// TIA Portal V20 export
FUNCTION_BLOCK "CallEquipment"   // FB64, LAD
TITLE = CallEquipment
// This block includes all general functions, checks and logik that is needed in the entire unit. E.g. general releases and system wide functionalities like air, pressure and power handling as well as general reaction to events.
// stored: IsIECCheckEnabled true, MemoryReserve 100, Namespace Unit1.Em6, SetENOAutomatically true
   VAR_INPUT
      ZoneOperationEnable { ExternalWritable := 'False'} : "LWONIK_typeSafetyZoneManualOperation";
   END_VAR
   VAR_IN_OUT
      unitStatus : "LAF_typeUnitStatus";   // Current unit status o be used in this EM
      emFeedback : "LUC_typeEmFeedback";   // Feedback of the EM to the Unit
      unitAlarmDB : "LAF_typeAlarms";   // Summarized EM Alarms for the Unit
   END_VAR
   VAR
      InstHotPressLeftSequence { ExternalWritable := 'False'} : "Unit1.Em6.Sequence_1_HotPressLeft";
      instHotPressLeftHomeJob1 { ExternalWritable := 'False'} : "LAF_SelectJob";
      instHotPressLeftLoadJob2 { ExternalWritable := 'False'} : "LAF_SelectJob";
      instHotPressLeftInspectionJob3 { ExternalWritable := 'False'} : "LAF_SelectJob";
      instHotPressLeftUnloadJob4 { ExternalWritable := 'False'} : "LAF_SelectJob";
      instCmHotPressLeftSafetyPin { ExternalWritable := 'False'} : "LBC_DigitalSignalCn";
      instCmHotPressLeftJRDetect { ExternalWritable := 'False'} : "LBC_DigitalSignalCn";
      instCmHotPressLeftStageLiftFrontUpDown { ExternalWritable := 'False'} : "LBC_TwoWayActuatorCn";
      instCmHotPressLeftStageLiftRearUpDown { ExternalWritable := 'False'} : "LBC_TwoWayActuatorCn";
      instCmHotPressLeftStageLiftAllUpDown { ExternalWritable := 'False'} : "LBC_TwoWayActuatorCn";
      instCmHotPressLeftTemperature { ExternalWritable := 'False'} : "LER_Heater";
      instCmHotPressLeftServoPress { ExternalWritable := 'False'} : "LER_ServoPress";
      instCmHotPressLeftHistroy { ExternalWritable := 'False'} : "LER_ServoPressHistory";
      instManageAlarms { ExternalWritable := 'False'} : "LAF_ManageAlarms";
      instEventsPFE { ExternalWritable := 'False'} : "Unit1.Em6.EventsPFE";
      statUnitStatus { ExternalWritable := 'False'} : "LAF_typeUnitStatus";   // Unit Status that is used in this project
   END_VAR
   VAR RETAIN
      statPartData { ExternalWritable := 'False'} : "LER_typePartData";
   END_VAR
   VAR
      statDataDelete { ExternalWritable := 'False'} : "LER_typePartData";
      statHistoryDeleteData { ExternalWritable := 'False'} : "LER_typeServoPressHistory";
      statClock { ExternalWritable := 'False'} : "LAF_typeGlobalClockMem";
      statTonTime { ExternalWritable := 'False'} : Array[0..999] of TON_TIME;
      statTofTime { ExternalWritable := 'False'} : Array[0..9] of TOF_TIME;
      statPulse { ExternalWritable := 'False'} : Array[0..999] of Bool;
      statNomalMode { ExternalWritable := 'False'} : Bool;
      statEnableManualCmds { ExternalWritable := 'False'} : Bool;
      statDoorOpenTemperature { ExternalWritable := 'False'} : "Safety.typeHotPressTempOk";
      statRunTemperature { ExternalWritable := 'False'} : Bool;
      "*** Interlock TwoWay ***" { S7_SetPoint := 'True'} : "LER_Axis_Homing";
      instCmHotPressLeftStageLiftFrontUpDownInterlock { S7_SetPoint := 'True'} : Array[0..2] of "LER_Actuator";
      instCmHotPressLeftStageLiftRearUpDownInterlock { S7_SetPoint := 'True'} : Array[0..2] of "LER_Actuator";
      instCmHotPressLeftStageLiftAllUpDownInterlock { S7_SetPoint := 'True'} : Array[0..2] of "LER_Actuator";
      HotPressLeftStageLiftFrontUpDown_Inpos : Array[0..2] of Struct
         "Int" : Array[1..10] of Bool;
      END_STRUCT;
      HotPressLeftStageLiftRearUpDown_Inpos : Array[0..2] of Struct
         "Int" : Array[1..10] of Bool;
      END_STRUCT;
      HotPressLeftStageLiftAllUpDown_Inpos : Array[0..2] of Struct
         "Int" : Array[1..10] of Bool;
      END_STRUCT;
      citi_Ptrig : Array[0..20] of Bool;
      citiTon : Array[0..20] of TON_TIME;
      citi : Time;
      citiTest : Array[0..20] of Bool;
      statReal : Array[0..9] of Real;
      instPFERecipe { S7_SetPoint := 'True'} : "Unit1.Em6.EventsPFE_Recipe";
   END_VAR
   VAR_TEMP
      tempRET_VAL : Array[0..99] of Int;
      tempScInProduction : Bool;   // Mode Production and StateComplete
      tempScNoProduction : Bool;   // Mode Manual and StateComplete
      tempPlaceReq : Bool;   // Request placing to TRPnPRight
      tempInspecReq : Bool;
      tempPickReq : Bool;   // Request Pick to TRPnPRight
   END_VAR
   VAR CONSTANT
      delayTime : Time := T#3s;
      TRUE : Bool := TRUE;
      FALSE : Bool := FALSE;
      NO_JOB : DInt;
      Stacker1 : Char := 'A';
      Stacker2 : Char := 'B';
   END_VAR
   VAR_TEMP   // added for the SCL form of the ladder/FBD networks
      _w1 : Bool;
      _w2 : Bool;
      _w3 : Bool;
      _w4 : Bool;
      _w5 : Bool;
      _w6 : Bool;
      _w7 : Bool;
   END_VAR
BEGIN

REGION Network 1: BLOCK INFO HEADER
   // (company) / (C) Copyright (year)
   // ---------------------------------------------------------------------------------
   // Title:                             (Title of this block)
   // Comment/Function: (that is implemented in the block)
   // Library/Family:           (that the source is dedicated to)
   // Author:                        (department / person in charge / contact)
   // Target System:          (test system with FW version)
   // Engineering:              TIA Portal (SW version)
   // Restrictions:               (OB types, etc.)
   // Requirements:           (hardware, technological package, etc.)
   // ---------------------------------------------------------------------------------
   // Change log table:
   // Version          | Date             | Signature      | Expert in charge  | Changes applied ------------------------|----------------------|-------------------------|--------------------------------|-----------------------
   // 001.000.000 | yyyy-mm-dd | 0x00000000 | (name of expert) | First released version
END_REGION

REGION Network 2: DESCRIPTION
   // This is a template block provided by the Automation Framework. It can be used to create an own project.
   // The Block Info Header is prepared to put in your own data.
   // Description of the block could be added here and the docu created by Code2Docu.
END_REGION

REGION Network 3: Simulation
   // If simulation is active on a global level, inherit this status and set simulation active in this unit also. Information is written to DB ControlNodes, from where it is distributed to the equipmemt modules.
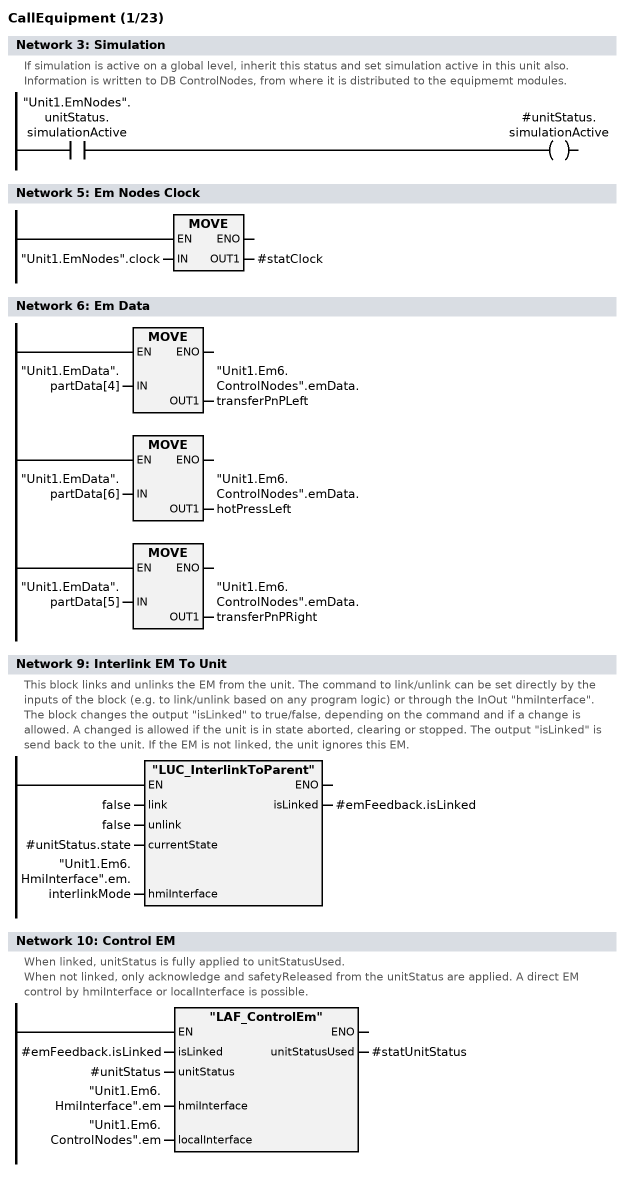
   RUNG wire#powerrail
      Contact( "Unit1.EmNodes".unitStatus.simulationActive )
      Coil( #unitStatus.simulationActive )
   END_RUNG
   // the same network as SCL:
   #unitStatus.simulationActive := "Unit1.EmNodes".unitStatus.simulationActive;
END_REGION

REGION Network 4: ******************** Unit Input ********************
END_REGION

REGION Network 5: Em Nodes Clock
   RUNG wire#powerrail
      Move(in := "Unit1.EmNodes".clock, out1 => #statClock)
   END_RUNG
   // the same network as SCL:
   #statClock := "Unit1.EmNodes".clock;
END_REGION

REGION Network 6: Em Data
   RUNG wire#powerrail
      Move(in := "Unit1.EmData".partData[4], out1 => "Unit1.Em6.ControlNodes".emData.transferPnPLeft)
   END_RUNG
   RUNG wire#powerrail
      Move(in := "Unit1.EmData".partData[6], out1 => "Unit1.Em6.ControlNodes".emData.hotPressLeft)
   END_RUNG
   RUNG wire#powerrail
      Move(in := "Unit1.EmData".partData[5], out1 => "Unit1.Em6.ControlNodes".emData.transferPnPRight)
   END_RUNG
   // the same network as SCL:
   "Unit1.Em6.ControlNodes".emData.transferPnPLeft := "Unit1.EmData".partData[4];
   "Unit1.Em6.ControlNodes".emData.hotPressLeft := "Unit1.EmData".partData[6];
   "Unit1.Em6.ControlNodes".emData.transferPnPRight := "Unit1.EmData".partData[5];
END_REGION

REGION Network 8: ******************** Equipment Control ********************
END_REGION

REGION Network 9: Interlink EM To Unit
   // This block links and unlinks the EM from the unit. The command to link/unlink can be set directly by the inputs of the block (e.g. to link/unlink based on any program logic) or through the InOut "hmiInterface". The block changes the output "isLinked" to true/false, depending on the command and if a change is allowed. A changed is allowed if the unit is in state aborted, clearing or stopped. The output "isLinked" is send back to the unit. If the EM is not linked, the unit ignores this EM.
   RUNG wire#powerrail
      "LUC_InterlinkToParent"(link := false, unlink := false, currentState := #unitStatus.state, hmiInterface := "Unit1.Em6.HmiInterface".em.interlinkMode, isLinked => #emFeedback.isLinked)
   END_RUNG
   // the same network as SCL:
   "LUC_InterlinkToParent"(link := false,
                           unlink := false,
                           currentState := #unitStatus.state,
                           hmiInterface := "Unit1.Em6.HmiInterface".em.interlinkMode,
                           isLinked => #emFeedback.isLinked);
END_REGION

REGION Network 10: Control EM
   // When linked, unitStatus is fully applied to unitStatusUsed.
   // When not linked, only acknowledge and safetyReleased from the unitStatus are applied. A direct EM control by hmiInterface or localInterface is possible.
   RUNG wire#powerrail
      "LAF_ControlEm"(isLinked := #emFeedback.isLinked, unitStatus := #unitStatus, hmiInterface := "Unit1.Em6.HmiInterface".em, localInterface := "Unit1.Em6.ControlNodes".em, unitStatusUsed => #statUnitStatus)
   END_RUNG
   // the same network as SCL:
   "LAF_ControlEm"(isLinked := #emFeedback.isLinked,
                   unitStatus := #unitStatus,
                   hmiInterface := "Unit1.Em6.HmiInterface".em,
                   localInterface := "Unit1.Em6.ControlNodes".em,
                   unitStatusUsed => #statUnitStatus);
END_REGION

REGION Network 11: EnableManualCmds
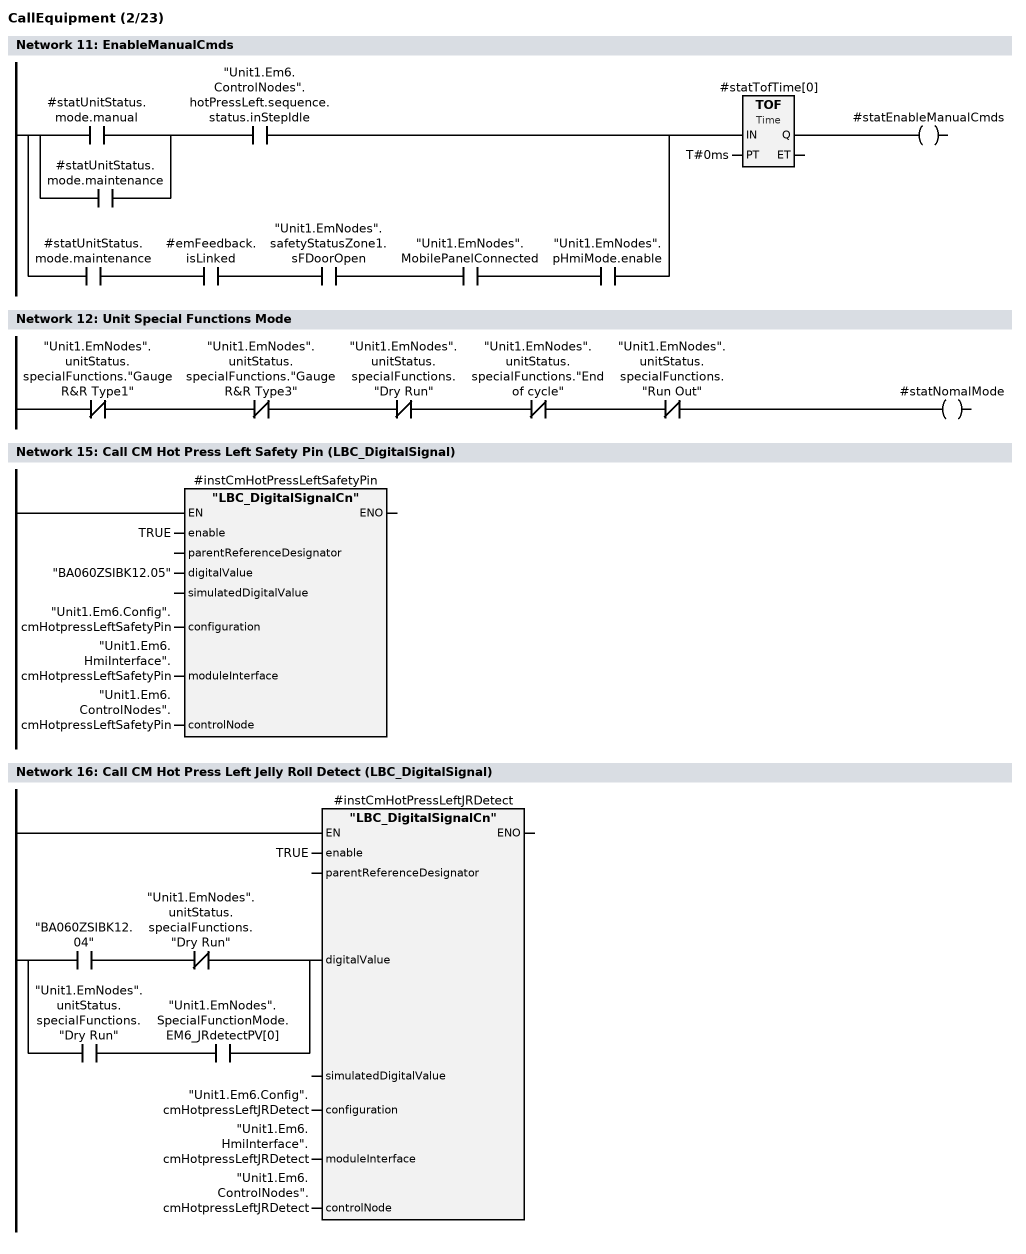
   RUNG wire#powerrail
      Contact( #statUnitStatus.mode.manual )
      wire#w1
      Contact( "Unit1.Em6.ControlNodes".hotPressLeft.sequence.status.inStepIdle )
      wire#w2
      { S7_Templates := "time_type := Time" } #statTofTime[0].TOF(pt := T#0ms, et =>)
      Coil( #statEnableManualCmds )
   END_RUNG
   RUNG wire#powerrail
      Contact( #statUnitStatus.mode.maintenance )
   END_RUNG wire#w1
   RUNG wire#powerrail
      Contact( #statUnitStatus.mode.maintenance )
      Contact( #emFeedback.isLinked )
      Contact( "Unit1.EmNodes".safetyStatusZone1.sFDoorOpen )
      Contact( "Unit1.EmNodes".MobilePanelConnected )
      Contact( "Unit1.EmNodes".pHmiMode.enable )
   END_RUNG wire#w2
   // the same network as SCL:
   #statTofTime[0].TOF(IN := ((#statUnitStatus.mode.manual OR #statUnitStatus.mode.maintenance) AND "Unit1.Em6.ControlNodes".hotPressLeft.sequence.status.inStepIdle) OR (#statUnitStatus.mode.maintenance AND #emFeedback.isLinked AND "Unit1.EmNodes".safetyStatusZone1.sFDoorOpen AND "Unit1.EmNodes".MobilePanelConnected AND "Unit1.EmNodes".pHmiMode.enable),
                       PT := T#0ms);
   #statEnableManualCmds := #statTofTime[0].Q;
END_REGION

REGION Network 12: Unit Special Functions Mode
   RUNG wire#powerrail
      I_Contact( "Unit1.EmNodes".unitStatus.specialFunctions."Gauge R&R Type1" )
      I_Contact( "Unit1.EmNodes".unitStatus.specialFunctions."Gauge R&R Type3" )
      I_Contact( "Unit1.EmNodes".unitStatus.specialFunctions."Dry Run" )
      I_Contact( "Unit1.EmNodes".unitStatus.specialFunctions."End of cycle" )
      I_Contact( "Unit1.EmNodes".unitStatus.specialFunctions."Run Out" )
      Coil( #statNomalMode )
   END_RUNG
   // the same network as SCL:
   #statNomalMode := NOT "Unit1.EmNodes".unitStatus.specialFunctions."Gauge R&R Type1" AND NOT "Unit1.EmNodes".unitStatus.specialFunctions."Gauge R&R Type3" AND NOT "Unit1.EmNodes".unitStatus.specialFunctions."Dry Run" AND NOT "Unit1.EmNodes".unitStatus.specialFunctions."End of cycle" AND NOT "Unit1.EmNodes".unitStatus.specialFunctions."Run Out";
END_REGION

REGION Network 14: ******************** Control Modules (Sensors) ********************
   // Call control modules that are sensors before the em logic (jobs and sequence), so that the latest value is used in the logic.
END_REGION

REGION Network 15: Call CM Hot Press Left Safety Pin (LBC_DigitalSignal)
   RUNG wire#powerrail
      #instCmHotPressLeftSafetyPin(enable := TRUE, parentReferenceDesignator :=, digitalValue := "BA060ZSIBK12.05", simulatedDigitalValue :=, configuration := "Unit1.Em6.Config".cmHotpressLeftSafetyPin, moduleInterface := "Unit1.Em6.HmiInterface".cmHotpressLeftSafetyPin, controlNode := "Unit1.Em6.ControlNodes".cmHotpressLeftSafetyPin)
   END_RUNG
   // the same network as SCL:
   #instCmHotPressLeftSafetyPin(enable := TRUE,   // "LBC_DigitalSignalCn"
                           digitalValue := "BA060ZSIBK12.05",
                           configuration := "Unit1.Em6.Config".cmHotpressLeftSafetyPin,
                           moduleInterface := "Unit1.Em6.HmiInterface".cmHotpressLeftSafetyPin,
                           controlNode := "Unit1.Em6.ControlNodes".cmHotpressLeftSafetyPin);
END_REGION

REGION Network 16: Call CM Hot Press Left Jelly Roll Detect (LBC_DigitalSignal)
   RUNG wire#powerrail
      #instCmHotPressLeftJRDetect(digitalValue := wire#w1, enable := TRUE, parentReferenceDesignator :=, simulatedDigitalValue :=, configuration := "Unit1.Em6.Config".cmHotpressLeftJRDetect, moduleInterface := "Unit1.Em6.HmiInterface".cmHotpressLeftJRDetect, controlNode := "Unit1.Em6.ControlNodes".cmHotpressLeftJRDetect)
   END_RUNG
   RUNG wire#powerrail
      Contact( "BA060ZSIBK12.04" )
      I_Contact( "Unit1.EmNodes".unitStatus.specialFunctions."Dry Run" )
   END_RUNG wire#w1
   RUNG wire#powerrail
      Contact( "Unit1.EmNodes".unitStatus.specialFunctions."Dry Run" )
      Contact( "Unit1.EmNodes".SpecialFunctionMode.EM6_JRdetectPV[0] )
   END_RUNG wire#w1
   // the same network as SCL:
   #instCmHotPressLeftJRDetect(enable := TRUE,   // "LBC_DigitalSignalCn"
                           digitalValue := ("BA060ZSIBK12.04" AND NOT "Unit1.EmNodes".unitStatus.specialFunctions."Dry Run") OR ("Unit1.EmNodes".unitStatus.specialFunctions."Dry Run" AND "Unit1.EmNodes".SpecialFunctionMode.EM6_JRdetectPV[0]),
                           configuration := "Unit1.Em6.Config".cmHotpressLeftJRDetect,
                           moduleInterface := "Unit1.Em6.HmiInterface".cmHotpressLeftJRDetect,
                           controlNode := "Unit1.Em6.ControlNodes".cmHotpressLeftJRDetect);
END_REGION

REGION Network 18: ******************** Equipment Logic ********************
END_REGION

REGION Network 19: Map Unit Status To Sequence Status
   // This block maps the unit status to the seuqnce status. Thus, it controls the sequence depending on the unit status. E.g. it sets the sequence to automatic when the unit state is in productions. This blocks work perfectly with the sequences provided in the AF. 
   // This typed block (MapUnitStatusToSequence) could be adjusted to specific application requirements or if other, user-defined sequences are used.
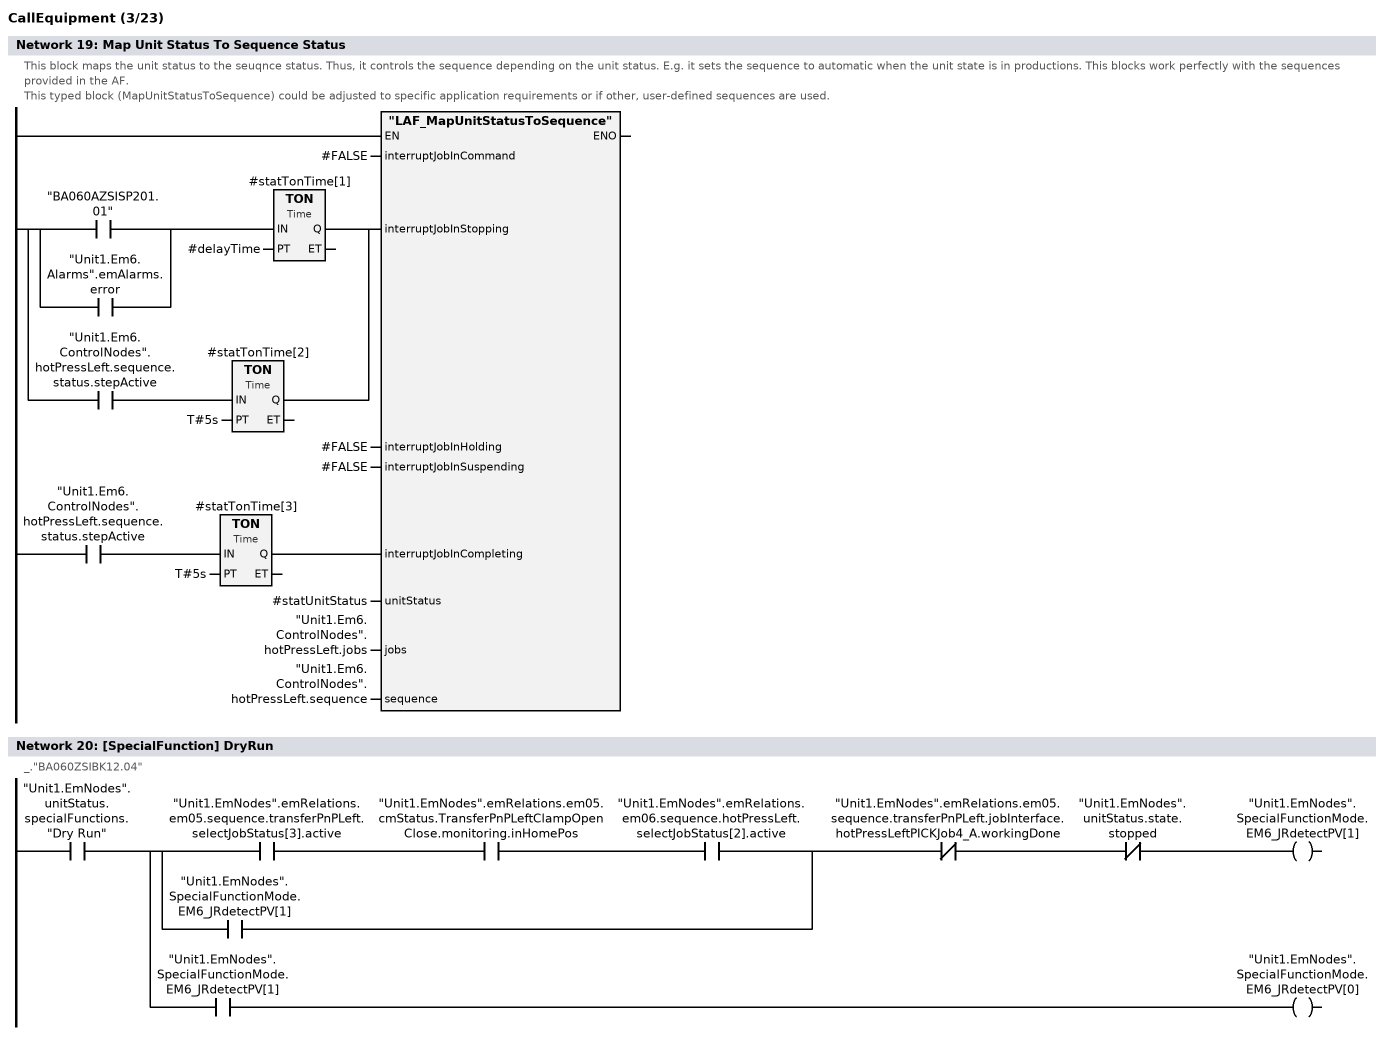
   RUNG wire#powerrail
      "LAF_MapUnitStatusToSequence"(interruptJobInStopping := wire#w2, interruptJobInCompleting := wire#w3, interruptJobInCommand := #FALSE, interruptJobInHolding := #FALSE, interruptJobInSuspending := #FALSE, unitStatus := #statUnitStatus, jobs := "Unit1.Em6.ControlNodes".hotPressLeft.jobs, sequence := "Unit1.Em6.ControlNodes".hotPressLeft.sequence)
   END_RUNG
   RUNG wire#powerrail
      Contact( "BA060AZSISP201.01" )
      wire#w1
      { S7_Templates := "time_type := Time" } #statTonTime[1].TON(pt := #delayTime, et =>)
   END_RUNG wire#w2
   RUNG wire#powerrail
      Contact( "Unit1.Em6.Alarms".emAlarms.error )
   END_RUNG wire#w1
   RUNG wire#powerrail
      Contact( "Unit1.Em6.ControlNodes".hotPressLeft.sequence.status.stepActive )
      { S7_Templates := "time_type := Time" } #statTonTime[2].TON(pt := T#5s, et =>)
   END_RUNG wire#w2
   RUNG wire#powerrail
      Contact( "Unit1.Em6.ControlNodes".hotPressLeft.sequence.status.stepActive )
      { S7_Templates := "time_type := Time" } #statTonTime[3].TON(pt := T#5s, et =>)
   END_RUNG wire#w3
   // the same network as SCL:
   #statTonTime[1].TON(IN := "BA060AZSISP201.01" OR "Unit1.Em6.Alarms".emAlarms.error, PT := #delayTime);
   #_w1 := #statTonTime[1].Q;
   #statTonTime[2].TON(IN := "Unit1.Em6.ControlNodes".hotPressLeft.sequence.status.stepActive, PT := T#5s);
   #_w2 := #_w1 OR #statTonTime[2].Q;
   #statTonTime[3].TON(IN := "Unit1.Em6.ControlNodes".hotPressLeft.sequence.status.stepActive, PT := T#5s);
   "LAF_MapUnitStatusToSequence"(interruptJobInCommand := #FALSE,
                           interruptJobInStopping := #_w2,
                           interruptJobInHolding := #FALSE,
                           interruptJobInSuspending := #FALSE,
                           interruptJobInCompleting := #statTonTime[3].Q,
                           unitStatus := #statUnitStatus,
                           jobs := "Unit1.Em6.ControlNodes".hotPressLeft.jobs,
                           sequence := "Unit1.Em6.ControlNodes".hotPressLeft.sequence);
END_REGION

REGION Network 20: [SpecialFunction] DryRun
   // _."BA060ZSIBK12.04"
   RUNG wire#powerrail
      Contact( "Unit1.EmNodes".unitStatus.specialFunctions."Dry Run" )
      wire#w1
      Contact( "Unit1.EmNodes".emRelations.em05.sequence.transferPnPLeft.selectJobStatus[3].active )
      Contact( "Unit1.EmNodes".emRelations.em05.cmStatus.TransferPnPLeftClampOpenClose.monitoring.inHomePos )
      Contact( "Unit1.EmNodes".emRelations.em06.sequence.hotPressLeft.selectJobStatus[2].active )
      wire#w2
      I_Contact( "Unit1.EmNodes".emRelations.em05.sequence.transferPnPLeft.jobInterface.hotPressLeftPICKJob4_A.workingDone )
      I_Contact( "Unit1.EmNodes".unitStatus.state.stopped )
      Coil( "Unit1.EmNodes".SpecialFunctionMode.EM6_JRdetectPV[1] )
   END_RUNG
   RUNG wire#w1
      Contact( "Unit1.EmNodes".SpecialFunctionMode.EM6_JRdetectPV[1] )
   END_RUNG wire#w2
   RUNG wire#w1
      Contact( "Unit1.EmNodes".SpecialFunctionMode.EM6_JRdetectPV[1] )
      Coil( "Unit1.EmNodes".SpecialFunctionMode.EM6_JRdetectPV[0] )
   END_RUNG
   // the same network as SCL:
   "Unit1.EmNodes".SpecialFunctionMode.EM6_JRdetectPV[1] := "Unit1.EmNodes".unitStatus.specialFunctions."Dry Run" AND (("Unit1.EmNodes".emRelations.em05.sequence.transferPnPLeft.selectJobStatus[3].active AND "Unit1.EmNodes".emRelations.em05.cmStatus.TransferPnPLeftClampOpenClose.monitoring.inHomePos AND "Unit1.EmNodes".emRelations.em06.sequence.hotPressLeft.selectJobStatus[2].active) OR "Unit1.EmNodes".SpecialFunctionMode.EM6_JRdetectPV[1]) AND NOT "Unit1.EmNodes".emRelations.em05.sequence.transferPnPLeft.jobInterface.hotPressLeftPICKJob4_A.workingDone AND NOT "Unit1.EmNodes".unitStatus.state.stopped;
   "Unit1.EmNodes".SpecialFunctionMode.EM6_JRdetectPV[0] := "Unit1.EmNodes".unitStatus.specialFunctions."Dry Run" AND "Unit1.EmNodes".SpecialFunctionMode.EM6_JRdetectPV[1];
END_REGION

REGION Network 22: [Job] Hot Press Left Select Job
   // Configure here when the jobs of the sequence should be started. More jobs could be added.
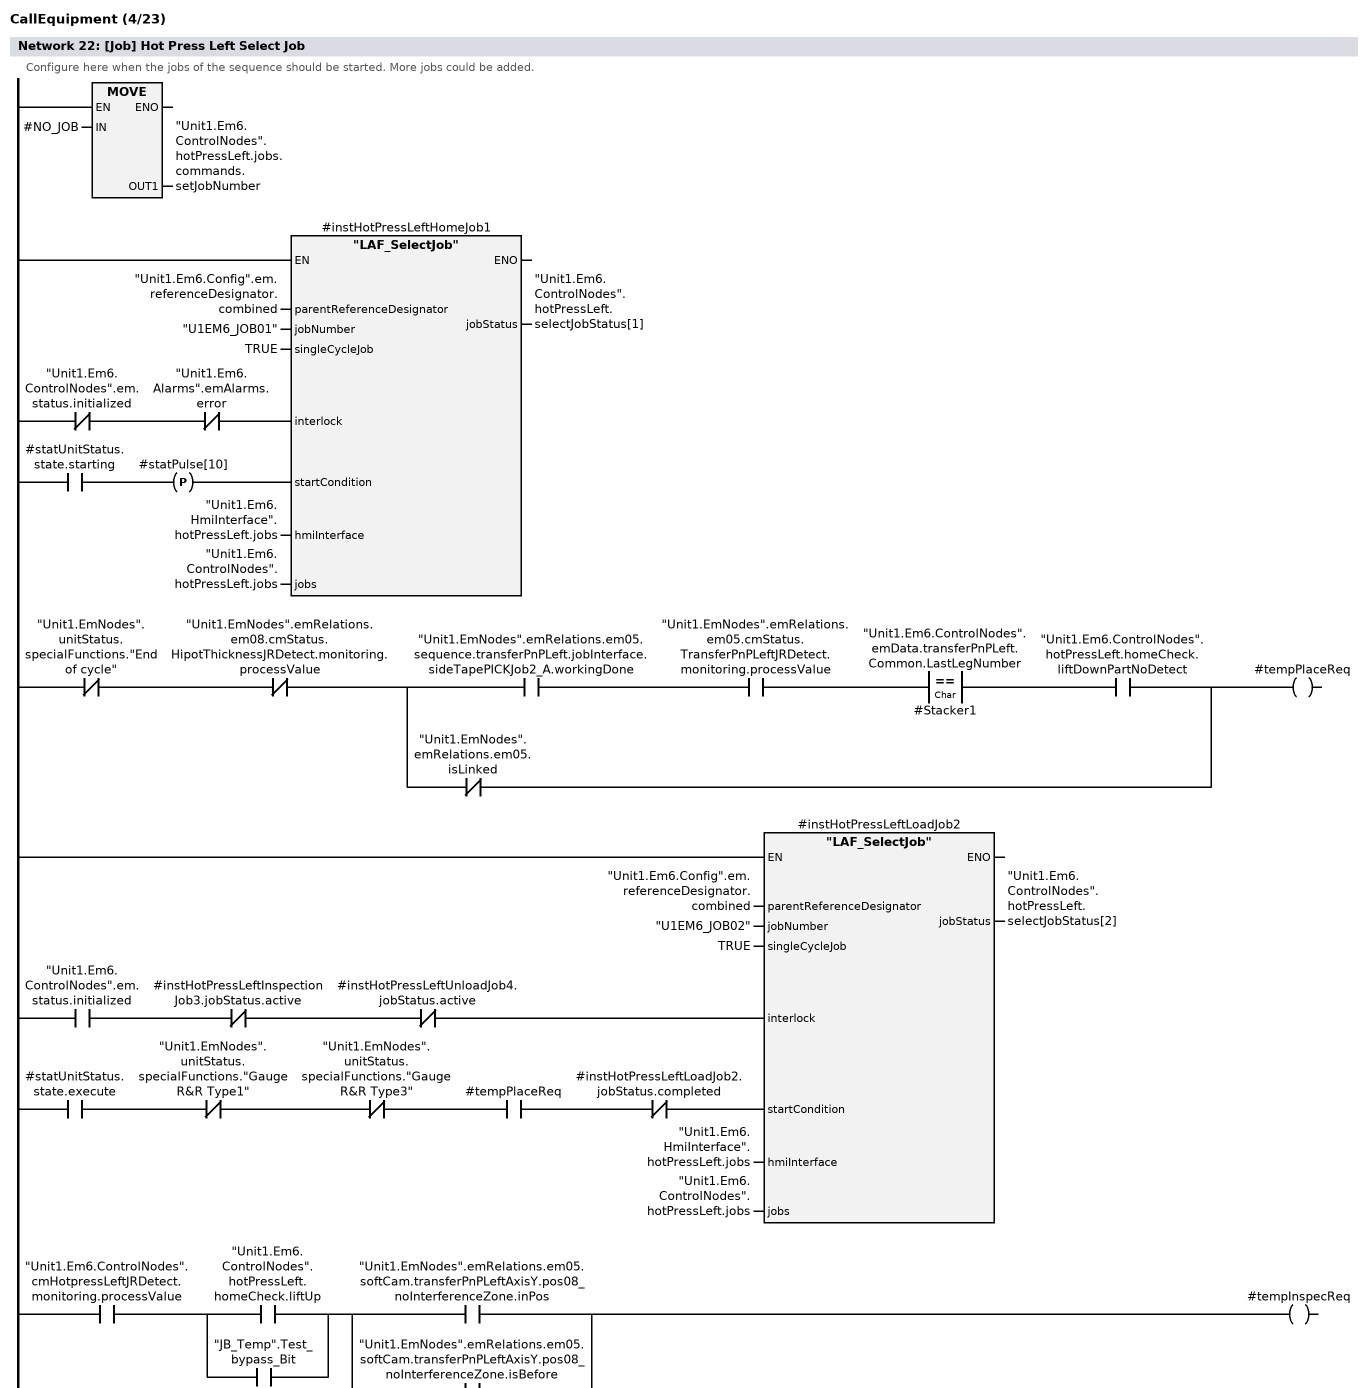
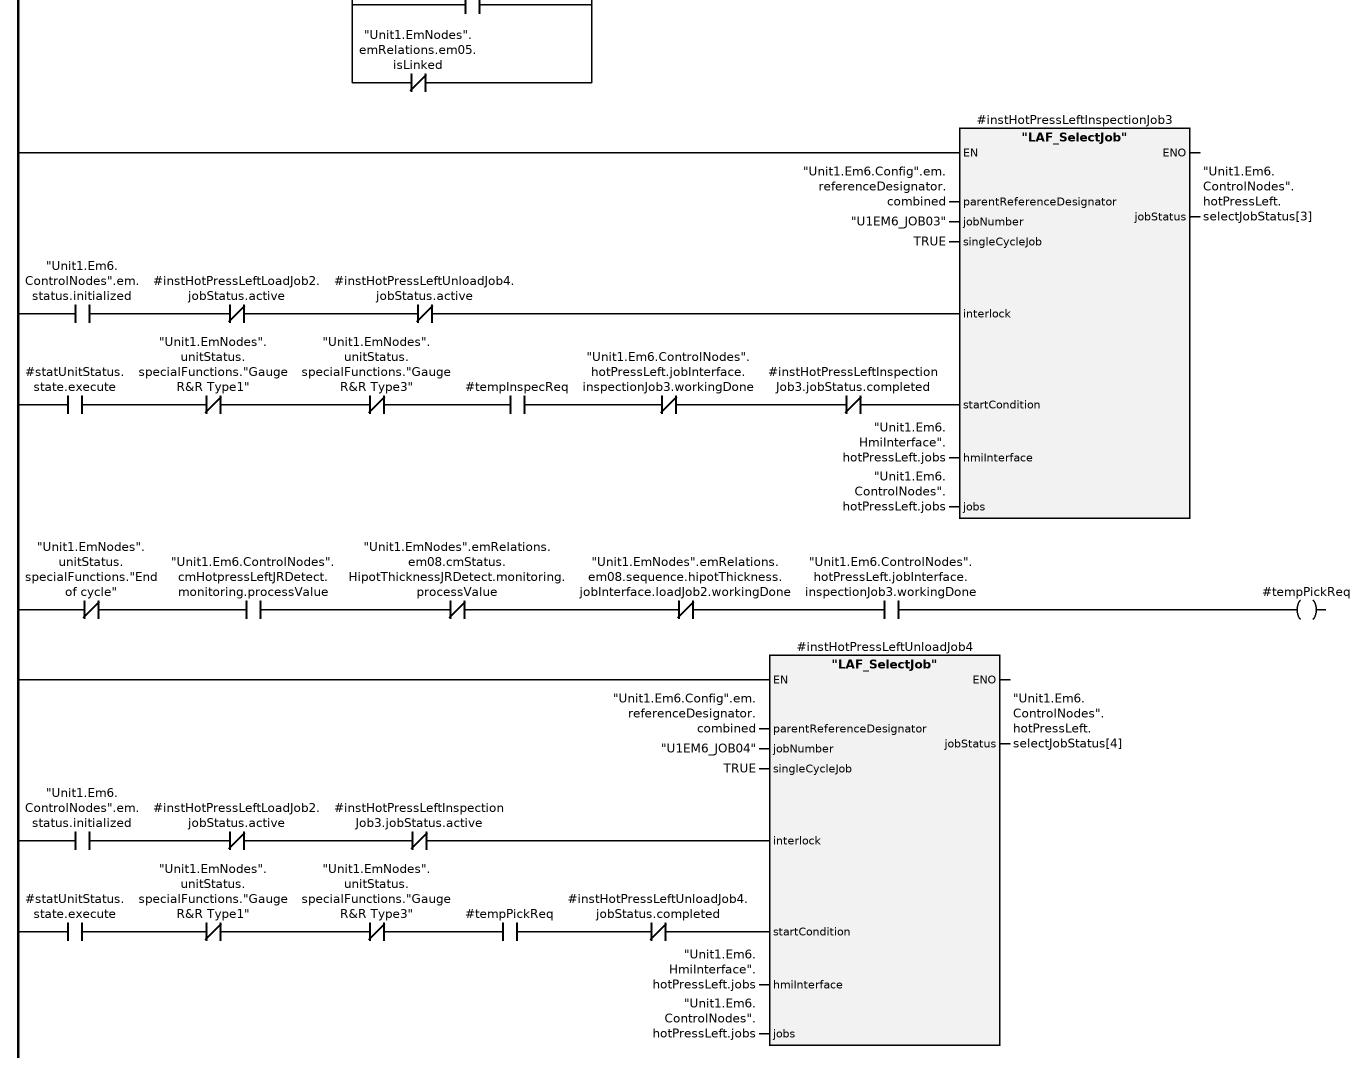
   RUNG wire#powerrail
      Move(in := #NO_JOB, out1 => "Unit1.Em6.ControlNodes".hotPressLeft.jobs.commands.setJobNumber)
   END_RUNG
   RUNG wire#powerrail
      #instHotPressLeftHomeJob1(interlock := wire#w1, startCondition := wire#w2, parentReferenceDesignator := "Unit1.Em6.Config".em.referenceDesignator.combined, jobNumber := "U1EM6_JOB01", singleCycleJob := TRUE, hmiInterface := "Unit1.Em6.HmiInterface".hotPressLeft.jobs, jobs := "Unit1.Em6.ControlNodes".hotPressLeft.jobs, jobStatus => "Unit1.Em6.ControlNodes".hotPressLeft.selectJobStatus[1])
   END_RUNG
   RUNG wire#powerrail
      I_Contact( "Unit1.Em6.ControlNodes".em.status.initialized )
      I_Contact( "Unit1.Em6.Alarms".emAlarms.error )
   END_RUNG wire#w1
   RUNG wire#powerrail
      Contact( #statUnitStatus.state.starting )
      P_Trig( #statPulse[10] )
   END_RUNG wire#w2
   RUNG wire#powerrail
      I_Contact( "Unit1.EmNodes".unitStatus.specialFunctions."End of cycle" )
      I_Contact( "Unit1.EmNodes".emRelations.em08.cmStatus.HipotThicknessJRDetect.monitoring.processValue )
      wire#w3
      Contact( "Unit1.EmNodes".emRelations.em05.sequence.transferPnPLeft.jobInterface.sideTapePICKJob2_A.workingDone )
      Contact( "Unit1.EmNodes".emRelations.em05.cmStatus.TransferPnPLeftJRDetect.monitoring.processValue )
      { S7_Templates := "SrcType := Char" } EQ_Contact(in1 := "Unit1.Em6.ControlNodes".emData.transferPnPLeft.Common.LastLegNumber, in2 := #Stacker1)
      Contact( "Unit1.Em6.ControlNodes".hotPressLeft.homeCheck.liftDownPartNoDetect )
      wire#w4
      Coil( #tempPlaceReq )
   END_RUNG
   RUNG wire#w3
      I_Contact( "Unit1.EmNodes".emRelations.em05.isLinked )
   END_RUNG wire#w4
   RUNG wire#powerrail
      #instHotPressLeftLoadJob2(interlock := wire#w5, startCondition := wire#w6, parentReferenceDesignator := "Unit1.Em6.Config".em.referenceDesignator.combined, jobNumber := "U1EM6_JOB02", singleCycleJob := TRUE, hmiInterface := "Unit1.Em6.HmiInterface".hotPressLeft.jobs, jobs := "Unit1.Em6.ControlNodes".hotPressLeft.jobs, jobStatus => "Unit1.Em6.ControlNodes".hotPressLeft.selectJobStatus[2])
   END_RUNG
   RUNG wire#powerrail
      Contact( "Unit1.Em6.ControlNodes".em.status.initialized )
      I_Contact( #instHotPressLeftInspectionJob3.jobStatus.active )
      I_Contact( #instHotPressLeftUnloadJob4.jobStatus.active )
   END_RUNG wire#w5
   RUNG wire#powerrail
      Contact( #statUnitStatus.state.execute )
      I_Contact( "Unit1.EmNodes".unitStatus.specialFunctions."Gauge R&R Type1" )
      I_Contact( "Unit1.EmNodes".unitStatus.specialFunctions."Gauge R&R Type3" )
      Contact( #tempPlaceReq )
      I_Contact( #instHotPressLeftLoadJob2.jobStatus.completed )
   END_RUNG wire#w6
   RUNG wire#powerrail
      Contact( "Unit1.Em6.ControlNodes".cmHotpressLeftJRDetect.monitoring.processValue )
      wire#w7
      Contact( "Unit1.Em6.ControlNodes".hotPressLeft.homeCheck.liftUp )
      wire#w8
      Contact( "Unit1.EmNodes".emRelations.em05.softCam.transferPnPLeftAxisY.pos08_noInterferenceZone.inPos )
      wire#w9
      Coil( #tempInspecReq )
   END_RUNG
   RUNG wire#w7
      Contact( "JB_Temp".Test_bypass_Bit )
   END_RUNG wire#w8
   RUNG wire#w8
      Contact( "Unit1.EmNodes".emRelations.em05.softCam.transferPnPLeftAxisY.pos08_noInterferenceZone.isBefore )
   END_RUNG wire#w9
   RUNG wire#w8
      I_Contact( "Unit1.EmNodes".emRelations.em05.isLinked )
   END_RUNG wire#w9
   RUNG wire#powerrail
      #instHotPressLeftInspectionJob3(interlock := wire#w10, startCondition := wire#w11, parentReferenceDesignator := "Unit1.Em6.Config".em.referenceDesignator.combined, jobNumber := "U1EM6_JOB03", singleCycleJob := TRUE, hmiInterface := "Unit1.Em6.HmiInterface".hotPressLeft.jobs, jobs := "Unit1.Em6.ControlNodes".hotPressLeft.jobs, jobStatus => "Unit1.Em6.ControlNodes".hotPressLeft.selectJobStatus[3])
   END_RUNG
   RUNG wire#powerrail
      Contact( "Unit1.Em6.ControlNodes".em.status.initialized )
      I_Contact( #instHotPressLeftLoadJob2.jobStatus.active )
      I_Contact( #instHotPressLeftUnloadJob4.jobStatus.active )
   END_RUNG wire#w10
   RUNG wire#powerrail
      Contact( #statUnitStatus.state.execute )
      I_Contact( "Unit1.EmNodes".unitStatus.specialFunctions."Gauge R&R Type1" )
      I_Contact( "Unit1.EmNodes".unitStatus.specialFunctions."Gauge R&R Type3" )
      Contact( #tempInspecReq )
      I_Contact( "Unit1.Em6.ControlNodes".hotPressLeft.jobInterface.inspectionJob3.workingDone )
      I_Contact( #instHotPressLeftInspectionJob3.jobStatus.completed )
   END_RUNG wire#w11
   RUNG wire#powerrail
      I_Contact( "Unit1.EmNodes".unitStatus.specialFunctions."End of cycle" )
      Contact( "Unit1.Em6.ControlNodes".cmHotpressLeftJRDetect.monitoring.processValue )
      I_Contact( "Unit1.EmNodes".emRelations.em08.cmStatus.HipotThicknessJRDetect.monitoring.processValue )
      I_Contact( "Unit1.EmNodes".emRelations.em08.sequence.hipotThickness.jobInterface.loadJob2.workingDone )
      Contact( "Unit1.Em6.ControlNodes".hotPressLeft.jobInterface.inspectionJob3.workingDone )
      Coil( #tempPickReq )
   END_RUNG
   RUNG wire#powerrail
      #instHotPressLeftUnloadJob4(interlock := wire#w12, startCondition := wire#w13, parentReferenceDesignator := "Unit1.Em6.Config".em.referenceDesignator.combined, jobNumber := "U1EM6_JOB04", singleCycleJob := TRUE, hmiInterface := "Unit1.Em6.HmiInterface".hotPressLeft.jobs, jobs := "Unit1.Em6.ControlNodes".hotPressLeft.jobs, jobStatus => "Unit1.Em6.ControlNodes".hotPressLeft.selectJobStatus[4])
   END_RUNG
   RUNG wire#powerrail
      Contact( "Unit1.Em6.ControlNodes".em.status.initialized )
      I_Contact( #instHotPressLeftLoadJob2.jobStatus.active )
      I_Contact( #instHotPressLeftInspectionJob3.jobStatus.active )
   END_RUNG wire#w12
   RUNG wire#powerrail
      Contact( #statUnitStatus.state.execute )
      I_Contact( "Unit1.EmNodes".unitStatus.specialFunctions."Gauge R&R Type1" )
      I_Contact( "Unit1.EmNodes".unitStatus.specialFunctions."Gauge R&R Type3" )
      Contact( #tempPickReq )
      I_Contact( #instHotPressLeftUnloadJob4.jobStatus.completed )
   END_RUNG wire#w13
   // the same network as SCL:
   "Unit1.Em6.ControlNodes".hotPressLeft.jobs.commands.setJobNumber := #NO_JOB;
   #_w1 := #statUnitStatus.state.starting AND NOT #statPulse[10];   // rising edge
   #statPulse[10] := #statUnitStatus.state.starting;
   #instHotPressLeftHomeJob1(parentReferenceDesignator := "Unit1.Em6.Config".em.referenceDesignator.combined,   // "LAF_SelectJob"
                           jobNumber := "U1EM6_JOB01",
                           singleCycleJob := TRUE,
                           interlock := NOT "Unit1.Em6.ControlNodes".em.status.initialized AND NOT "Unit1.Em6.Alarms".emAlarms.error,
                           startCondition := #_w1,
                           hmiInterface := "Unit1.Em6.HmiInterface".hotPressLeft.jobs,
                           jobs := "Unit1.Em6.ControlNodes".hotPressLeft.jobs,
                           jobStatus => "Unit1.Em6.ControlNodes".hotPressLeft.selectJobStatus[1]);
   #tempPlaceReq := NOT "Unit1.EmNodes".unitStatus.specialFunctions."End of cycle" AND NOT "Unit1.EmNodes".emRelations.em08.cmStatus.HipotThicknessJRDetect.monitoring.processValue AND (("Unit1.EmNodes".emRelations.em05.sequence.transferPnPLeft.jobInterface.sideTapePICKJob2_A.workingDone AND "Unit1.EmNodes".emRelations.em05.cmStatus.TransferPnPLeftJRDetect.monitoring.processValue AND ("Unit1.Em6.ControlNodes".emData.transferPnPLeft.Common.LastLegNumber = #Stacker1) AND "Unit1.Em6.ControlNodes".hotPressLeft.homeCheck.liftDownPartNoDetect) OR NOT "Unit1.EmNodes".emRelations.em05.isLinked);
   #instHotPressLeftLoadJob2(parentReferenceDesignator := "Unit1.Em6.Config".em.referenceDesignator.combined,   // "LAF_SelectJob"
                           jobNumber := "U1EM6_JOB02",
                           singleCycleJob := TRUE,
                           interlock := "Unit1.Em6.ControlNodes".em.status.initialized AND NOT #instHotPressLeftInspectionJob3.jobStatus.active AND NOT #instHotPressLeftUnloadJob4.jobStatus.active,
                           startCondition := #statUnitStatus.state.execute AND NOT "Unit1.EmNodes".unitStatus.specialFunctions."Gauge R&R Type1" AND NOT "Unit1.EmNodes".unitStatus.specialFunctions."Gauge R&R Type3" AND #tempPlaceReq AND NOT #instHotPressLeftLoadJob2.jobStatus.completed,
                           hmiInterface := "Unit1.Em6.HmiInterface".hotPressLeft.jobs,
                           jobs := "Unit1.Em6.ControlNodes".hotPressLeft.jobs,
                           jobStatus => "Unit1.Em6.ControlNodes".hotPressLeft.selectJobStatus[2]);
   #tempInspecReq := "Unit1.Em6.ControlNodes".cmHotpressLeftJRDetect.monitoring.processValue AND ("Unit1.Em6.ControlNodes".hotPressLeft.homeCheck.liftUp OR "JB_Temp".Test_bypass_Bit) AND ("Unit1.EmNodes".emRelations.em05.softCam.transferPnPLeftAxisY.pos08_noInterferenceZone.inPos OR "Unit1.EmNodes".emRelations.em05.softCam.transferPnPLeftAxisY.pos08_noInterferenceZone.isBefore OR NOT "Unit1.EmNodes".emRelations.em05.isLinked);
   #instHotPressLeftInspectionJob3(parentReferenceDesignator := "Unit1.Em6.Config".em.referenceDesignator.combined,   // "LAF_SelectJob"
                           jobNumber := "U1EM6_JOB03",
                           singleCycleJob := TRUE,
                           interlock := "Unit1.Em6.ControlNodes".em.status.initialized AND NOT #instHotPressLeftLoadJob2.jobStatus.active AND NOT #instHotPressLeftUnloadJob4.jobStatus.active,
                           startCondition := #statUnitStatus.state.execute AND NOT "Unit1.EmNodes".unitStatus.specialFunctions."Gauge R&R Type1" AND NOT "Unit1.EmNodes".unitStatus.specialFunctions."Gauge R&R Type3" AND #tempInspecReq AND NOT "Unit1.Em6.ControlNodes".hotPressLeft.jobInterface.inspectionJob3.workingDone AND NOT #instHotPressLeftInspectionJob3.jobStatus.completed,
                           hmiInterface := "Unit1.Em6.HmiInterface".hotPressLeft.jobs,
                           jobs := "Unit1.Em6.ControlNodes".hotPressLeft.jobs,
                           jobStatus => "Unit1.Em6.ControlNodes".hotPressLeft.selectJobStatus[3]);
   #tempPickReq := NOT "Unit1.EmNodes".unitStatus.specialFunctions."End of cycle" AND "Unit1.Em6.ControlNodes".cmHotpressLeftJRDetect.monitoring.processValue AND NOT "Unit1.EmNodes".emRelations.em08.cmStatus.HipotThicknessJRDetect.monitoring.processValue AND NOT "Unit1.EmNodes".emRelations.em08.sequence.hipotThickness.jobInterface.loadJob2.workingDone AND "Unit1.Em6.ControlNodes".hotPressLeft.jobInterface.inspectionJob3.workingDone;
   #instHotPressLeftUnloadJob4(parentReferenceDesignator := "Unit1.Em6.Config".em.referenceDesignator.combined,   // "LAF_SelectJob"
                           jobNumber := "U1EM6_JOB04",
                           singleCycleJob := TRUE,
                           interlock := "Unit1.Em6.ControlNodes".em.status.initialized AND NOT #instHotPressLeftLoadJob2.jobStatus.active AND NOT #instHotPressLeftInspectionJob3.jobStatus.active,
                           startCondition := #statUnitStatus.state.execute AND NOT "Unit1.EmNodes".unitStatus.specialFunctions."Gauge R&R Type1" AND NOT "Unit1.EmNodes".unitStatus.specialFunctions."Gauge R&R Type3" AND #tempPickReq AND NOT #instHotPressLeftUnloadJob4.jobStatus.completed,
                           hmiInterface := "Unit1.Em6.HmiInterface".hotPressLeft.jobs,
                           jobs := "Unit1.Em6.ControlNodes".hotPressLeft.jobs,
                           jobStatus => "Unit1.Em6.ControlNodes".hotPressLeft.selectJobStatus[4]);
END_REGION

REGION Network 23: Hot Press left Job Interface [Loading]
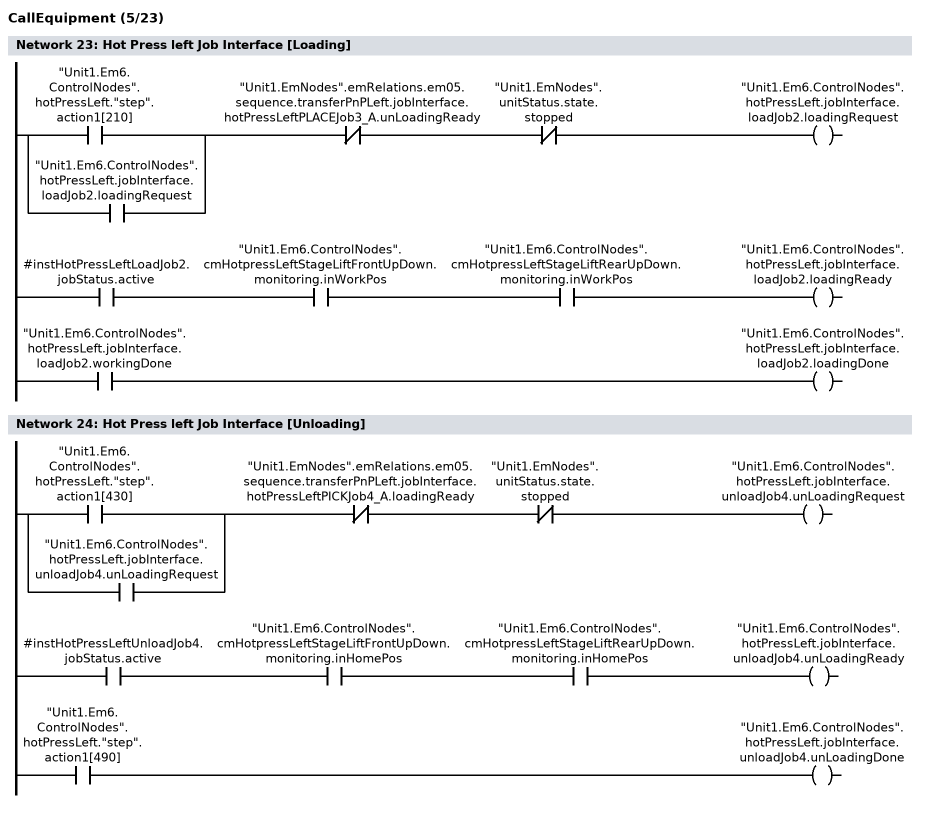
   RUNG wire#powerrail
      Contact( "Unit1.Em6.ControlNodes".hotPressLeft."step".action1[210] )
      wire#w1
      I_Contact( "Unit1.EmNodes".emRelations.em05.sequence.transferPnPLeft.jobInterface.hotPressLeftPLACEJob3_A.unLoadingReady )
      I_Contact( "Unit1.EmNodes".unitStatus.state.stopped )
      Coil( "Unit1.Em6.ControlNodes".hotPressLeft.jobInterface.loadJob2.loadingRequest )
   END_RUNG
   RUNG wire#powerrail
      Contact( "Unit1.Em6.ControlNodes".hotPressLeft.jobInterface.loadJob2.loadingRequest )
   END_RUNG wire#w1
   RUNG wire#powerrail
      Contact( #instHotPressLeftLoadJob2.jobStatus.active )
      Contact( "Unit1.Em6.ControlNodes".cmHotpressLeftStageLiftFrontUpDown.monitoring.inWorkPos )
      Contact( "Unit1.Em6.ControlNodes".cmHotpressLeftStageLiftRearUpDown.monitoring.inWorkPos )
      Coil( "Unit1.Em6.ControlNodes".hotPressLeft.jobInterface.loadJob2.loadingReady )
   END_RUNG
   RUNG wire#powerrail
      Contact( "Unit1.Em6.ControlNodes".hotPressLeft.jobInterface.loadJob2.workingDone )
      Coil( "Unit1.Em6.ControlNodes".hotPressLeft.jobInterface.loadJob2.loadingDone )
   END_RUNG
   // the same network as SCL:
   "Unit1.Em6.ControlNodes".hotPressLeft.jobInterface.loadJob2.loadingRequest := ("Unit1.Em6.ControlNodes".hotPressLeft."step".action1[210] OR "Unit1.Em6.ControlNodes".hotPressLeft.jobInterface.loadJob2.loadingRequest) AND NOT "Unit1.EmNodes".emRelations.em05.sequence.transferPnPLeft.jobInterface.hotPressLeftPLACEJob3_A.unLoadingReady AND NOT "Unit1.EmNodes".unitStatus.state.stopped;
   "Unit1.Em6.ControlNodes".hotPressLeft.jobInterface.loadJob2.loadingReady := #instHotPressLeftLoadJob2.jobStatus.active AND "Unit1.Em6.ControlNodes".cmHotpressLeftStageLiftFrontUpDown.monitoring.inWorkPos AND "Unit1.Em6.ControlNodes".cmHotpressLeftStageLiftRearUpDown.monitoring.inWorkPos;
   "Unit1.Em6.ControlNodes".hotPressLeft.jobInterface.loadJob2.loadingDone := "Unit1.Em6.ControlNodes".hotPressLeft.jobInterface.loadJob2.workingDone;
END_REGION

REGION Network 24: Hot Press left Job Interface [Unloading]
   RUNG wire#powerrail
      Contact( "Unit1.Em6.ControlNodes".hotPressLeft."step".action1[430] )
      wire#w1
      I_Contact( "Unit1.EmNodes".emRelations.em05.sequence.transferPnPLeft.jobInterface.hotPressLeftPICKJob4_A.loadingReady )
      I_Contact( "Unit1.EmNodes".unitStatus.state.stopped )
      Coil( "Unit1.Em6.ControlNodes".hotPressLeft.jobInterface.unloadJob4.unLoadingRequest )
   END_RUNG
   RUNG wire#powerrail
      Contact( "Unit1.Em6.ControlNodes".hotPressLeft.jobInterface.unloadJob4.unLoadingRequest )
   END_RUNG wire#w1
   RUNG wire#powerrail
      Contact( #instHotPressLeftUnloadJob4.jobStatus.active )
      Contact( "Unit1.Em6.ControlNodes".cmHotpressLeftStageLiftFrontUpDown.monitoring.inHomePos )
      Contact( "Unit1.Em6.ControlNodes".cmHotpressLeftStageLiftRearUpDown.monitoring.inHomePos )
      Coil( "Unit1.Em6.ControlNodes".hotPressLeft.jobInterface.unloadJob4.unLoadingReady )
   END_RUNG
   RUNG wire#powerrail
      Contact( "Unit1.Em6.ControlNodes".hotPressLeft."step".action1[490] )
      Coil( "Unit1.Em6.ControlNodes".hotPressLeft.jobInterface.unloadJob4.unLoadingDone )
   END_RUNG
   // the same network as SCL:
   "Unit1.Em6.ControlNodes".hotPressLeft.jobInterface.unloadJob4.unLoadingRequest := ("Unit1.Em6.ControlNodes".hotPressLeft."step".action1[430] OR "Unit1.Em6.ControlNodes".hotPressLeft.jobInterface.unloadJob4.unLoadingRequest) AND NOT "Unit1.EmNodes".emRelations.em05.sequence.transferPnPLeft.jobInterface.hotPressLeftPICKJob4_A.loadingReady AND NOT "Unit1.EmNodes".unitStatus.state.stopped;
   "Unit1.Em6.ControlNodes".hotPressLeft.jobInterface.unloadJob4.unLoadingReady := #instHotPressLeftUnloadJob4.jobStatus.active AND "Unit1.Em6.ControlNodes".cmHotpressLeftStageLiftFrontUpDown.monitoring.inHomePos AND "Unit1.Em6.ControlNodes".cmHotpressLeftStageLiftRearUpDown.monitoring.inHomePos;
   "Unit1.Em6.ControlNodes".hotPressLeft.jobInterface.unloadJob4.unLoadingDone := "Unit1.Em6.ControlNodes".hotPressLeft."step".action1[490];
END_REGION

REGION Network 25: Hot Press Left Job Interface Working Done
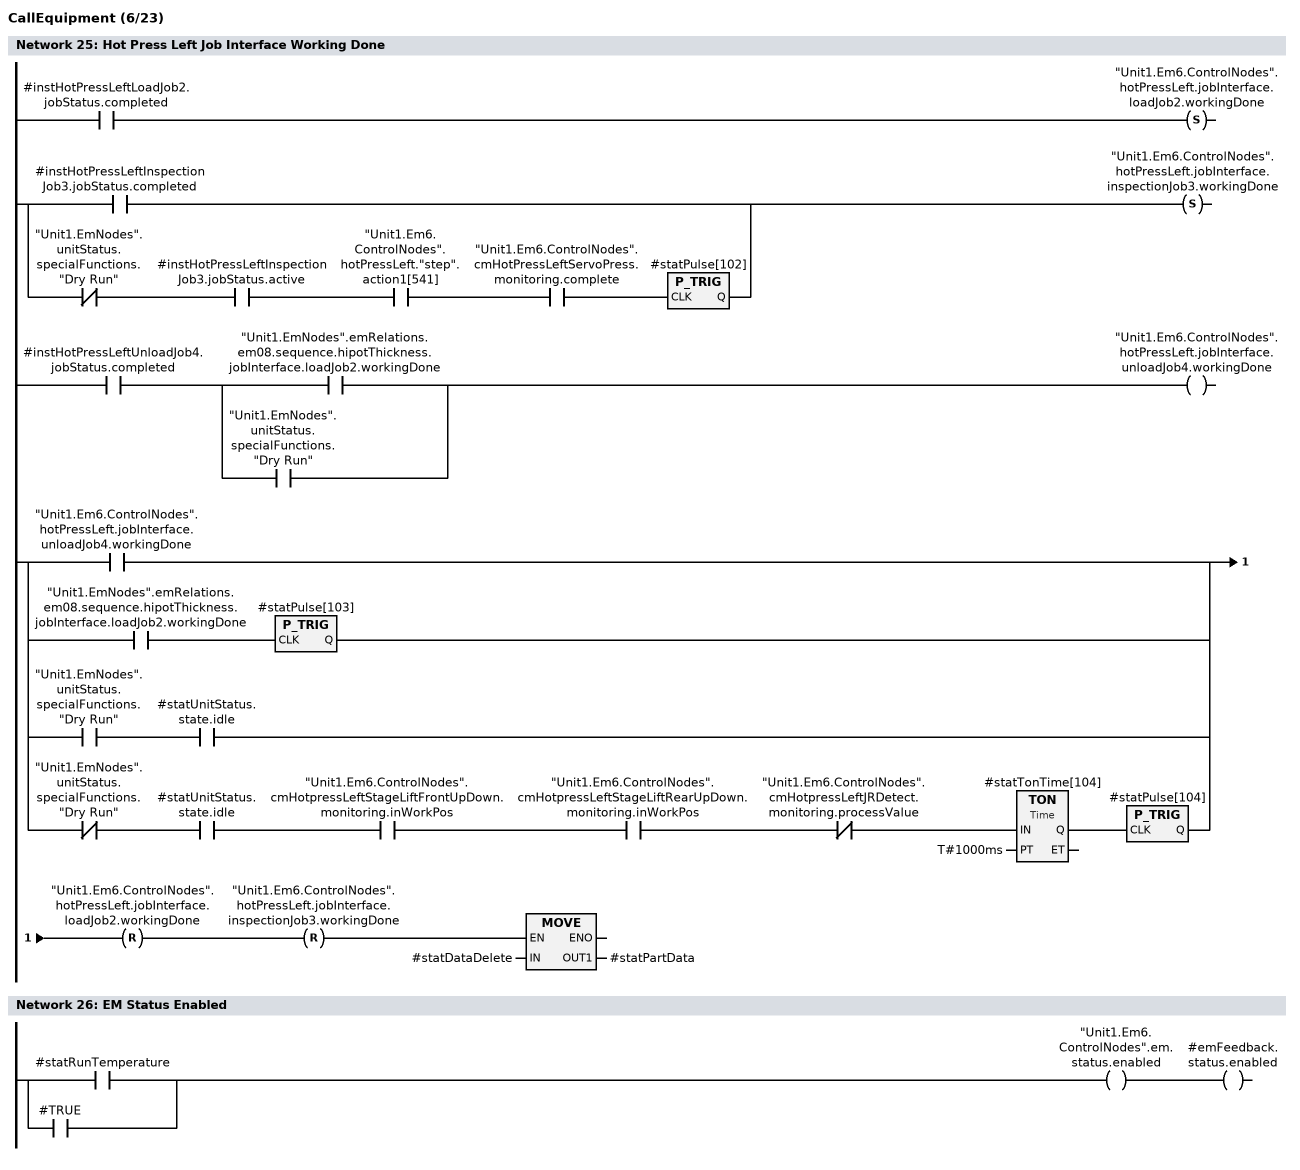
   RUNG wire#powerrail
      Contact( #instHotPressLeftLoadJob2.jobStatus.completed )
      S_Coil( "Unit1.Em6.ControlNodes".hotPressLeft.jobInterface.loadJob2.workingDone )
   END_RUNG
   RUNG wire#powerrail
      Contact( #instHotPressLeftInspectionJob3.jobStatus.completed )
      wire#w1
      S_Coil( "Unit1.Em6.ControlNodes".hotPressLeft.jobInterface.inspectionJob3.workingDone )
   END_RUNG
   RUNG wire#powerrail
      I_Contact( "Unit1.EmNodes".unitStatus.specialFunctions."Dry Run" )
      Contact( #instHotPressLeftInspectionJob3.jobStatus.active )
      Contact( "Unit1.Em6.ControlNodes".hotPressLeft."step".action1[541] )
      Contact( "Unit1.Em6.ControlNodes".cmHotPressLeftServoPress.monitoring.complete )
      P_Trig( #statPulse[102] )
   END_RUNG wire#w1
   RUNG wire#powerrail
      Contact( #instHotPressLeftUnloadJob4.jobStatus.completed )
      wire#w2
      Contact( "Unit1.EmNodes".emRelations.em08.sequence.hipotThickness.jobInterface.loadJob2.workingDone )
      wire#w3
      Coil( "Unit1.Em6.ControlNodes".hotPressLeft.jobInterface.unloadJob4.workingDone )
   END_RUNG
   RUNG wire#w2
      Contact( "Unit1.EmNodes".unitStatus.specialFunctions."Dry Run" )
   END_RUNG wire#w3
   RUNG wire#powerrail
      Contact( "Unit1.Em6.ControlNodes".hotPressLeft.jobInterface.unloadJob4.workingDone )
      wire#w4
      R_Coil( "Unit1.Em6.ControlNodes".hotPressLeft.jobInterface.loadJob2.workingDone )
      R_Coil( "Unit1.Em6.ControlNodes".hotPressLeft.jobInterface.inspectionJob3.workingDone )
      Move(in := #statDataDelete, out1 => #statPartData)
   END_RUNG
   RUNG wire#powerrail
      Contact( "Unit1.EmNodes".emRelations.em08.sequence.hipotThickness.jobInterface.loadJob2.workingDone )
      P_Trig( #statPulse[103] )
   END_RUNG wire#w4
   RUNG wire#powerrail
      Contact( "Unit1.EmNodes".unitStatus.specialFunctions."Dry Run" )
      Contact( #statUnitStatus.state.idle )
   END_RUNG wire#w4
   RUNG wire#powerrail
      I_Contact( "Unit1.EmNodes".unitStatus.specialFunctions."Dry Run" )
      Contact( #statUnitStatus.state.idle )
      Contact( "Unit1.Em6.ControlNodes".cmHotpressLeftStageLiftFrontUpDown.monitoring.inWorkPos )
      Contact( "Unit1.Em6.ControlNodes".cmHotpressLeftStageLiftRearUpDown.monitoring.inWorkPos )
      I_Contact( "Unit1.Em6.ControlNodes".cmHotpressLeftJRDetect.monitoring.processValue )
      { S7_Templates := "time_type := Time" } #statTonTime[104].TON(pt := T#1000ms, et =>)
      P_Trig( #statPulse[104] )
   END_RUNG wire#w4
   // the same network as SCL:
   IF #instHotPressLeftLoadJob2.jobStatus.completed THEN
       "Unit1.Em6.ControlNodes".hotPressLeft.jobInterface.loadJob2.workingDone := TRUE;
   END_IF;
   #_w1 := NOT "Unit1.EmNodes".unitStatus.specialFunctions."Dry Run" AND #instHotPressLeftInspectionJob3.jobStatus.active AND "Unit1.Em6.ControlNodes".hotPressLeft."step".action1[541] AND "Unit1.Em6.ControlNodes".cmHotPressLeftServoPress.monitoring.complete;
   #_w2 := #_w1 AND NOT #statPulse[102];   // rising edge
   #statPulse[102] := #_w1;
   IF #instHotPressLeftInspectionJob3.jobStatus.completed OR #_w2 THEN
       "Unit1.Em6.ControlNodes".hotPressLeft.jobInterface.inspectionJob3.workingDone := TRUE;
   END_IF;
   "Unit1.Em6.ControlNodes".hotPressLeft.jobInterface.unloadJob4.workingDone := #instHotPressLeftUnloadJob4.jobStatus.completed AND ("Unit1.EmNodes".emRelations.em08.sequence.hipotThickness.jobInterface.loadJob2.workingDone OR "Unit1.EmNodes".unitStatus.specialFunctions."Dry Run");
   #_w3 := "Unit1.EmNodes".emRelations.em08.sequence.hipotThickness.jobInterface.loadJob2.workingDone AND NOT #statPulse[103];   // rising edge
   #statPulse[103] := "Unit1.EmNodes".emRelations.em08.sequence.hipotThickness.jobInterface.loadJob2.workingDone;
   #statTonTime[104].TON(IN := NOT "Unit1.EmNodes".unitStatus.specialFunctions."Dry Run" AND #statUnitStatus.state.idle AND "Unit1.Em6.ControlNodes".cmHotpressLeftStageLiftFrontUpDown.monitoring.inWorkPos AND "Unit1.Em6.ControlNodes".cmHotpressLeftStageLiftRearUpDown.monitoring.inWorkPos AND NOT "Unit1.Em6.ControlNodes".cmHotpressLeftJRDetect.monitoring.processValue,
                         PT := T#1000ms);
   #_w4 := #statTonTime[104].Q AND NOT #statPulse[104];   // rising edge
   #statPulse[104] := #statTonTime[104].Q;
   IF "Unit1.Em6.ControlNodes".hotPressLeft.jobInterface.unloadJob4.workingDone OR #_w3 OR ("Unit1.EmNodes".unitStatus.specialFunctions."Dry Run" AND #statUnitStatus.state.idle) OR #_w4 THEN
       "Unit1.Em6.ControlNodes".hotPressLeft.jobInterface.loadJob2.workingDone := FALSE;
       "Unit1.Em6.ControlNodes".hotPressLeft.jobInterface.inspectionJob3.workingDone := FALSE;
       #statPartData := #statDataDelete;
   END_IF;
END_REGION

REGION Network 26: EM Status Enabled
   RUNG wire#powerrail
      Contact( #statRunTemperature )
      wire#w1
      Coil( "Unit1.Em6.ControlNodes".em.status.enabled )
      Coil( #emFeedback.status.enabled )
   END_RUNG
   RUNG wire#powerrail
      Contact( #TRUE )
   END_RUNG wire#w1
   // the same network as SCL:
   "Unit1.Em6.ControlNodes".em.status.enabled := #statRunTemperature OR #TRUE;
   #emFeedback.status.enabled := "Unit1.Em6.ControlNodes".em.status.enabled;
END_REGION

REGION Network 27: Set EM To Initialized
   // Set em to initialized here. Usually this is done when the initialization job is completed.
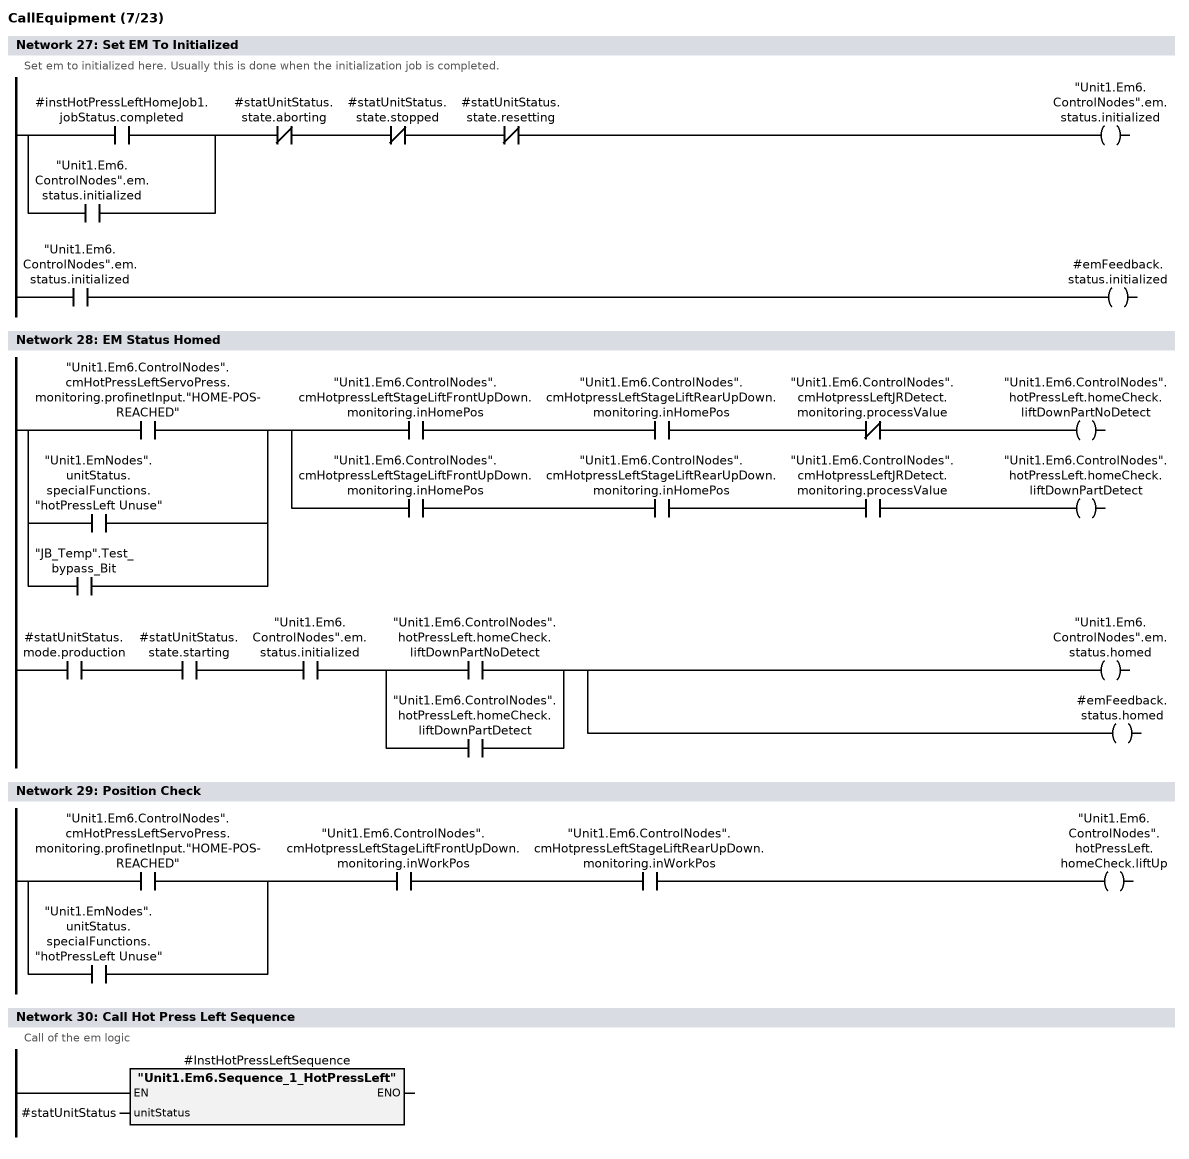
   RUNG wire#powerrail
      Contact( #instHotPressLeftHomeJob1.jobStatus.completed )
      wire#w1
      I_Contact( #statUnitStatus.state.aborting )
      I_Contact( #statUnitStatus.state.stopped )
      I_Contact( #statUnitStatus.state.resetting )
      Coil( "Unit1.Em6.ControlNodes".em.status.initialized )
   END_RUNG
   RUNG wire#powerrail
      Contact( "Unit1.Em6.ControlNodes".em.status.initialized )
   END_RUNG wire#w1
   RUNG wire#powerrail
      Contact( "Unit1.Em6.ControlNodes".em.status.initialized )
      Coil( #emFeedback.status.initialized )
   END_RUNG
   // the same network as SCL:
   "Unit1.Em6.ControlNodes".em.status.initialized := (#instHotPressLeftHomeJob1.jobStatus.completed OR "Unit1.Em6.ControlNodes".em.status.initialized) AND NOT #statUnitStatus.state.aborting AND NOT #statUnitStatus.state.stopped AND NOT #statUnitStatus.state.resetting;
   #emFeedback.status.initialized := "Unit1.Em6.ControlNodes".em.status.initialized;
END_REGION

REGION Network 28: EM Status Homed
   RUNG wire#powerrail
      Contact( "Unit1.Em6.ControlNodes".cmHotPressLeftServoPress.monitoring.profinetInput."HOME-POS-REACHED" )
      wire#w1
      Contact( "Unit1.Em6.ControlNodes".cmHotpressLeftStageLiftFrontUpDown.monitoring.inHomePos )
      Contact( "Unit1.Em6.ControlNodes".cmHotpressLeftStageLiftRearUpDown.monitoring.inHomePos )
      I_Contact( "Unit1.Em6.ControlNodes".cmHotpressLeftJRDetect.monitoring.processValue )
      Coil( "Unit1.Em6.ControlNodes".hotPressLeft.homeCheck.liftDownPartNoDetect )
   END_RUNG
   RUNG wire#powerrail
      Contact( "Unit1.EmNodes".unitStatus.specialFunctions."hotPressLeft Unuse" )
   END_RUNG wire#w1
   RUNG wire#powerrail
      Contact( "JB_Temp".Test_bypass_Bit )
   END_RUNG wire#w1
   RUNG wire#w1
      Contact( "Unit1.Em6.ControlNodes".cmHotpressLeftStageLiftFrontUpDown.monitoring.inHomePos )
      Contact( "Unit1.Em6.ControlNodes".cmHotpressLeftStageLiftRearUpDown.monitoring.inHomePos )
      Contact( "Unit1.Em6.ControlNodes".cmHotpressLeftJRDetect.monitoring.processValue )
      Coil( "Unit1.Em6.ControlNodes".hotPressLeft.homeCheck.liftDownPartDetect )
   END_RUNG
   RUNG wire#powerrail
      Contact( #statUnitStatus.mode.production )
      Contact( #statUnitStatus.state.starting )
      Contact( "Unit1.Em6.ControlNodes".em.status.initialized )
      wire#w2
      Contact( "Unit1.Em6.ControlNodes".hotPressLeft.homeCheck.liftDownPartNoDetect )
      wire#w3
      Coil( "Unit1.Em6.ControlNodes".em.status.homed )
   END_RUNG
   RUNG wire#w2
      Contact( "Unit1.Em6.ControlNodes".hotPressLeft.homeCheck.liftDownPartDetect )
   END_RUNG wire#w3
   RUNG wire#w3
      Coil( #emFeedback.status.homed )
   END_RUNG
   // the same network as SCL:
   #_w1 := "Unit1.Em6.ControlNodes".cmHotPressLeftServoPress.monitoring.profinetInput."HOME-POS-REACHED" OR "Unit1.EmNodes".unitStatus.specialFunctions."hotPressLeft Unuse" OR "JB_Temp".Test_bypass_Bit;
   "Unit1.Em6.ControlNodes".hotPressLeft.homeCheck.liftDownPartNoDetect := #_w1 AND "Unit1.Em6.ControlNodes".cmHotpressLeftStageLiftFrontUpDown.monitoring.inHomePos AND "Unit1.Em6.ControlNodes".cmHotpressLeftStageLiftRearUpDown.monitoring.inHomePos AND NOT "Unit1.Em6.ControlNodes".cmHotpressLeftJRDetect.monitoring.processValue;
   "Unit1.Em6.ControlNodes".hotPressLeft.homeCheck.liftDownPartDetect := #_w1 AND "Unit1.Em6.ControlNodes".cmHotpressLeftStageLiftFrontUpDown.monitoring.inHomePos AND "Unit1.Em6.ControlNodes".cmHotpressLeftStageLiftRearUpDown.monitoring.inHomePos AND "Unit1.Em6.ControlNodes".cmHotpressLeftJRDetect.monitoring.processValue;
   "Unit1.Em6.ControlNodes".em.status.homed := #statUnitStatus.mode.production AND #statUnitStatus.state.starting AND "Unit1.Em6.ControlNodes".em.status.initialized AND ("Unit1.Em6.ControlNodes".hotPressLeft.homeCheck.liftDownPartNoDetect OR "Unit1.Em6.ControlNodes".hotPressLeft.homeCheck.liftDownPartDetect);
   #emFeedback.status.homed := "Unit1.Em6.ControlNodes".em.status.homed;
END_REGION

REGION Network 29: Position Check
   RUNG wire#powerrail
      Contact( "Unit1.Em6.ControlNodes".cmHotPressLeftServoPress.monitoring.profinetInput."HOME-POS-REACHED" )
      wire#w1
      Contact( "Unit1.Em6.ControlNodes".cmHotpressLeftStageLiftFrontUpDown.monitoring.inWorkPos )
      Contact( "Unit1.Em6.ControlNodes".cmHotpressLeftStageLiftRearUpDown.monitoring.inWorkPos )
      Coil( "Unit1.Em6.ControlNodes".hotPressLeft.homeCheck.liftUp )
   END_RUNG
   RUNG wire#powerrail
      Contact( "Unit1.EmNodes".unitStatus.specialFunctions."hotPressLeft Unuse" )
   END_RUNG wire#w1
   // the same network as SCL:
   "Unit1.Em6.ControlNodes".hotPressLeft.homeCheck.liftUp := ("Unit1.Em6.ControlNodes".cmHotPressLeftServoPress.monitoring.profinetInput."HOME-POS-REACHED" OR "Unit1.EmNodes".unitStatus.specialFunctions."hotPressLeft Unuse") AND "Unit1.Em6.ControlNodes".cmHotpressLeftStageLiftFrontUpDown.monitoring.inWorkPos AND "Unit1.Em6.ControlNodes".cmHotpressLeftStageLiftRearUpDown.monitoring.inWorkPos;
END_REGION

REGION Network 30: Call Hot Press Left Sequence
   // Call of the em logic
   RUNG wire#powerrail
      #InstHotPressLeftSequence(unitStatus := #statUnitStatus)
   END_RUNG
   // the same network as SCL:
   #InstHotPressLeftSequence(unitStatus := #statUnitStatus);   // "Unit1.Em6.Sequence_1_HotPressLeft"
END_REGION

REGION Network 31: Hot Press Left Status
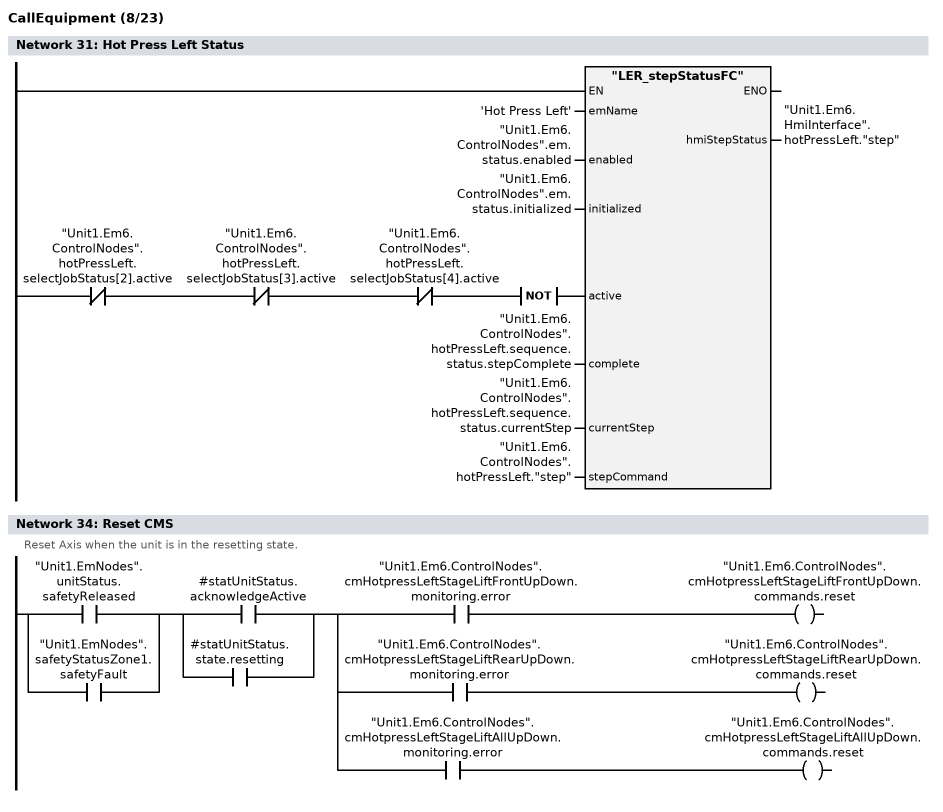
   RUNG wire#powerrail
      "LER_stepStatusFC"(active := wire#w1, emName := 'Hot Press Left', enabled := "Unit1.Em6.ControlNodes".em.status.enabled, initialized := "Unit1.Em6.ControlNodes".em.status.initialized, complete := "Unit1.Em6.ControlNodes".hotPressLeft.sequence.status.stepComplete, currentStep := "Unit1.Em6.ControlNodes".hotPressLeft.sequence.status.currentStep, stepCommand := "Unit1.Em6.ControlNodes".hotPressLeft."step", hmiStepStatus => "Unit1.Em6.HmiInterface".hotPressLeft."step")
   END_RUNG
   RUNG wire#powerrail
      I_Contact( "Unit1.Em6.ControlNodes".hotPressLeft.selectJobStatus[2].active )
      I_Contact( "Unit1.Em6.ControlNodes".hotPressLeft.selectJobStatus[3].active )
      I_Contact( "Unit1.Em6.ControlNodes".hotPressLeft.selectJobStatus[4].active )
      Not()
   END_RUNG wire#w1
   // the same network as SCL:
   "LER_stepStatusFC"(emName := 'Hot Press Left',
                      enabled := "Unit1.Em6.ControlNodes".em.status.enabled,
                      initialized := "Unit1.Em6.ControlNodes".em.status.initialized,
                      active := NOT (NOT "Unit1.Em6.ControlNodes".hotPressLeft.selectJobStatus[2].active AND NOT "Unit1.Em6.ControlNodes".hotPressLeft.selectJobStatus[3].active AND NOT "Unit1.Em6.ControlNodes".hotPressLeft.selectJobStatus[4].active),
                      complete := "Unit1.Em6.ControlNodes".hotPressLeft.sequence.status.stepComplete,
                      currentStep := "Unit1.Em6.ControlNodes".hotPressLeft.sequence.status.currentStep,
                      stepCommand := "Unit1.Em6.ControlNodes".hotPressLeft."step",
                      hmiStepStatus => "Unit1.Em6.HmiInterface".hotPressLeft."step");
END_REGION

REGION Network 33: ******************** Control Modules (TwoWayActuator) ********************
   // Call control modules that are actuators after the em logic (jobs and sequence), so that the latest commands are applied to the actuators.
END_REGION

REGION Network 34: Reset CMS
   // Reset Axis when the unit is in the resetting state.
   RUNG wire#powerrail
      Contact( "Unit1.EmNodes".unitStatus.safetyReleased )
      wire#w1
      Contact( #statUnitStatus.acknowledgeActive )
      wire#w2
      Contact( "Unit1.Em6.ControlNodes".cmHotpressLeftStageLiftFrontUpDown.monitoring.error )
      Coil( "Unit1.Em6.ControlNodes".cmHotpressLeftStageLiftFrontUpDown.commands.reset )
   END_RUNG
   RUNG wire#powerrail
      Contact( "Unit1.EmNodes".safetyStatusZone1.safetyFault )
   END_RUNG wire#w1
   RUNG wire#w1
      Contact( #statUnitStatus.state.resetting )
   END_RUNG wire#w2
   RUNG wire#w2
      Contact( "Unit1.Em6.ControlNodes".cmHotpressLeftStageLiftRearUpDown.monitoring.error )
      Coil( "Unit1.Em6.ControlNodes".cmHotpressLeftStageLiftRearUpDown.commands.reset )
   END_RUNG
   RUNG wire#w2
      Contact( "Unit1.Em6.ControlNodes".cmHotpressLeftStageLiftAllUpDown.monitoring.error )
      Coil( "Unit1.Em6.ControlNodes".cmHotpressLeftStageLiftAllUpDown.commands.reset )
   END_RUNG
   // the same network as SCL:
   #_w1 := ("Unit1.EmNodes".unitStatus.safetyReleased OR "Unit1.EmNodes".safetyStatusZone1.safetyFault) AND (#statUnitStatus.acknowledgeActive OR #statUnitStatus.state.resetting);
   "Unit1.Em6.ControlNodes".cmHotpressLeftStageLiftFrontUpDown.commands.reset := #_w1 AND "Unit1.Em6.ControlNodes".cmHotpressLeftStageLiftFrontUpDown.monitoring.error;
   "Unit1.Em6.ControlNodes".cmHotpressLeftStageLiftRearUpDown.commands.reset := #_w1 AND "Unit1.Em6.ControlNodes".cmHotpressLeftStageLiftRearUpDown.monitoring.error;
   "Unit1.Em6.ControlNodes".cmHotpressLeftStageLiftAllUpDown.commands.reset := #_w1 AND "Unit1.Em6.ControlNodes".cmHotpressLeftStageLiftAllUpDown.monitoring.error;
END_REGION

REGION Network 36: Hot Press Left Stage Lift Front Interlock Condition
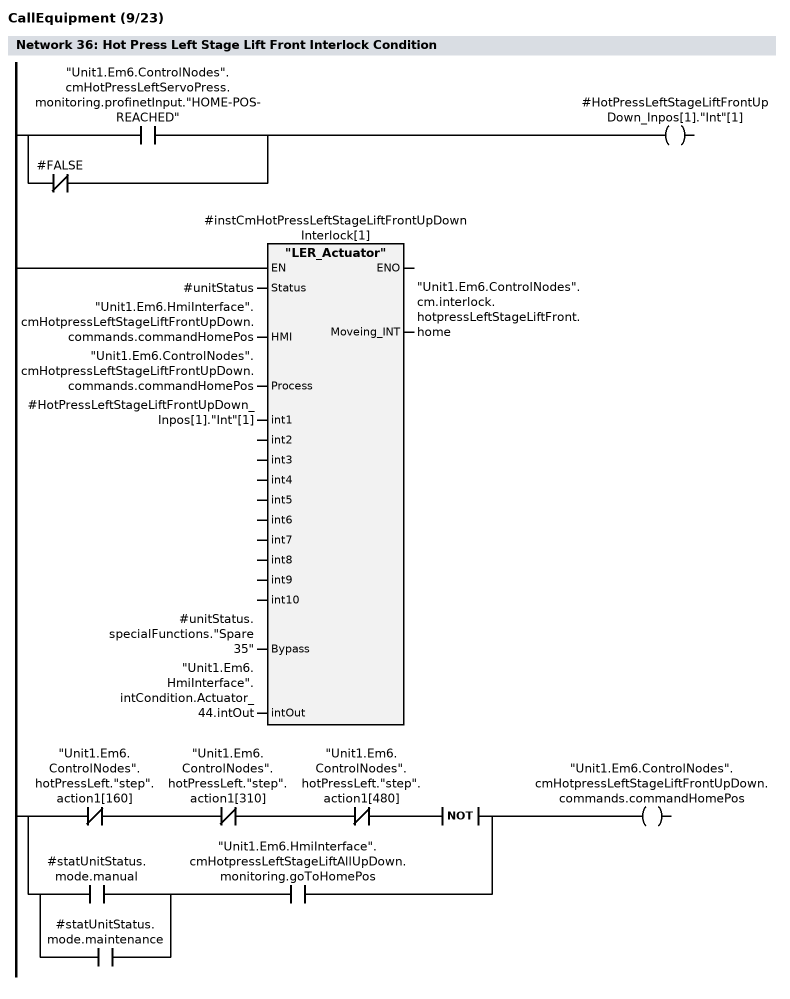
   RUNG wire#powerrail
      Contact( "Unit1.Em6.ControlNodes".cmHotPressLeftServoPress.monitoring.profinetInput."HOME-POS-REACHED" )
      wire#w1
      Coil( #HotPressLeftStageLiftFrontUpDown_Inpos[1]."Int"[1] )
   END_RUNG
   RUNG wire#powerrail
      I_Contact( #FALSE )
   END_RUNG wire#w1
   RUNG wire#powerrail
      #instCmHotPressLeftStageLiftFrontUpDownInterlock[1](Status := #unitStatus, HMI := "Unit1.Em6.HmiInterface".cmHotpressLeftStageLiftFrontUpDown.commands.commandHomePos, Process := "Unit1.Em6.ControlNodes".cmHotpressLeftStageLiftFrontUpDown.commands.commandHomePos, int1 := #HotPressLeftStageLiftFrontUpDown_Inpos[1]."Int"[1], int2 :=, int3 :=, int4 :=, int5 :=, int6 :=, int7 :=, int8 :=, int9 :=, int10 :=, Bypass := #unitStatus.specialFunctions."Spare 35", intOut := "Unit1.Em6.HmiInterface".intCondition.Actuator_44.intOut, Moveing_INT => "Unit1.Em6.ControlNodes".cm.interlock.hotpressLeftStageLiftFront.home)
   END_RUNG
   RUNG wire#powerrail
      I_Contact( "Unit1.Em6.ControlNodes".hotPressLeft."step".action1[160] )
      I_Contact( "Unit1.Em6.ControlNodes".hotPressLeft."step".action1[310] )
      I_Contact( "Unit1.Em6.ControlNodes".hotPressLeft."step".action1[480] )
      Not()
      wire#w2
      Coil( "Unit1.Em6.ControlNodes".cmHotpressLeftStageLiftFrontUpDown.commands.commandHomePos )
   END_RUNG
   RUNG wire#powerrail
      Contact( #statUnitStatus.mode.manual )
      wire#w3
      Contact( "Unit1.Em6.HmiInterface".cmHotpressLeftStageLiftAllUpDown.monitoring.goToHomePos )
   END_RUNG wire#w2
   RUNG wire#powerrail
      Contact( #statUnitStatus.mode.maintenance )
   END_RUNG wire#w3
   // the same network as SCL:
   #HotPressLeftStageLiftFrontUpDown_Inpos[1]."Int"[1] := "Unit1.Em6.ControlNodes".cmHotPressLeftServoPress.monitoring.profinetInput."HOME-POS-REACHED" OR NOT #FALSE;
   #instCmHotPressLeftStageLiftFrontUpDownInterlock[1](Status := #unitStatus,   // "LER_Actuator"
                           HMI := "Unit1.Em6.HmiInterface".cmHotpressLeftStageLiftFrontUpDown.commands.commandHomePos,
                           Process := "Unit1.Em6.ControlNodes".cmHotpressLeftStageLiftFrontUpDown.commands.commandHomePos,
                           int1 := #HotPressLeftStageLiftFrontUpDown_Inpos[1]."Int"[1],
                           Bypass := #unitStatus.specialFunctions."Spare 35",
                           intOut := "Unit1.Em6.HmiInterface".intCondition.Actuator_44.intOut,
                           Moveing_INT => "Unit1.Em6.ControlNodes".cm.interlock.hotpressLeftStageLiftFront.home);
   "Unit1.Em6.ControlNodes".cmHotpressLeftStageLiftFrontUpDown.commands.commandHomePos := NOT (NOT "Unit1.Em6.ControlNodes".hotPressLeft."step".action1[160] AND NOT "Unit1.Em6.ControlNodes".hotPressLeft."step".action1[310] AND NOT "Unit1.Em6.ControlNodes".hotPressLeft."step".action1[480]) OR ((#statUnitStatus.mode.manual OR #statUnitStatus.mode.maintenance) AND "Unit1.Em6.HmiInterface".cmHotpressLeftStageLiftAllUpDown.monitoring.goToHomePos);
END_REGION

REGION Network 37: Hot Press Left Stage Lift Front Commands
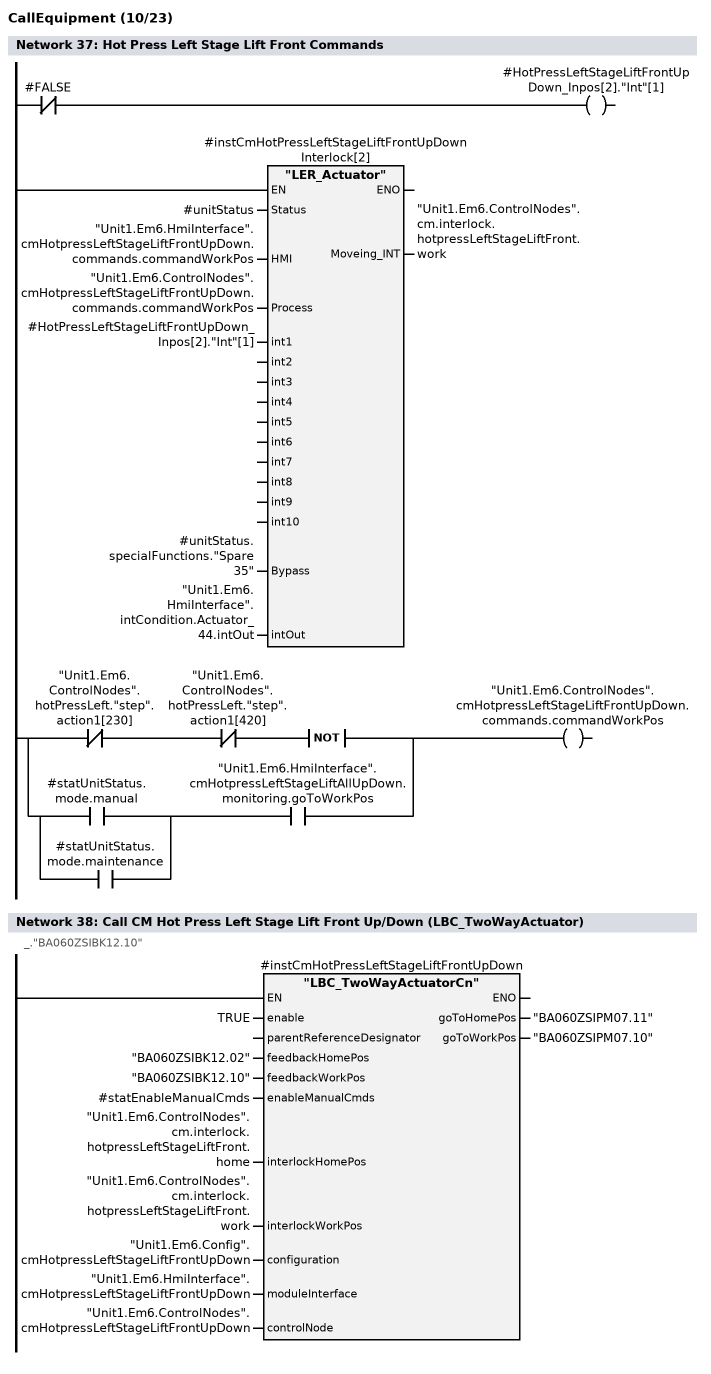
   RUNG wire#powerrail
      I_Contact( #FALSE )
      Coil( #HotPressLeftStageLiftFrontUpDown_Inpos[2]."Int"[1] )
   END_RUNG
   RUNG wire#powerrail
      #instCmHotPressLeftStageLiftFrontUpDownInterlock[2](Status := #unitStatus, HMI := "Unit1.Em6.HmiInterface".cmHotpressLeftStageLiftFrontUpDown.commands.commandWorkPos, Process := "Unit1.Em6.ControlNodes".cmHotpressLeftStageLiftFrontUpDown.commands.commandWorkPos, int1 := #HotPressLeftStageLiftFrontUpDown_Inpos[2]."Int"[1], int2 :=, int3 :=, int4 :=, int5 :=, int6 :=, int7 :=, int8 :=, int9 :=, int10 :=, Bypass := #unitStatus.specialFunctions."Spare 35", intOut := "Unit1.Em6.HmiInterface".intCondition.Actuator_44.intOut, Moveing_INT => "Unit1.Em6.ControlNodes".cm.interlock.hotpressLeftStageLiftFront.work)
   END_RUNG
   RUNG wire#powerrail
      I_Contact( "Unit1.Em6.ControlNodes".hotPressLeft."step".action1[230] )
      I_Contact( "Unit1.Em6.ControlNodes".hotPressLeft."step".action1[420] )
      Not()
      wire#w1
      Coil( "Unit1.Em6.ControlNodes".cmHotpressLeftStageLiftFrontUpDown.commands.commandWorkPos )
   END_RUNG
   RUNG wire#powerrail
      Contact( #statUnitStatus.mode.manual )
      wire#w2
      Contact( "Unit1.Em6.HmiInterface".cmHotpressLeftStageLiftAllUpDown.monitoring.goToWorkPos )
   END_RUNG wire#w1
   RUNG wire#powerrail
      Contact( #statUnitStatus.mode.maintenance )
   END_RUNG wire#w2
   // the same network as SCL:
   #HotPressLeftStageLiftFrontUpDown_Inpos[2]."Int"[1] := NOT #FALSE;
   #instCmHotPressLeftStageLiftFrontUpDownInterlock[2](Status := #unitStatus,   // "LER_Actuator"
                           HMI := "Unit1.Em6.HmiInterface".cmHotpressLeftStageLiftFrontUpDown.commands.commandWorkPos,
                           Process := "Unit1.Em6.ControlNodes".cmHotpressLeftStageLiftFrontUpDown.commands.commandWorkPos,
                           int1 := #HotPressLeftStageLiftFrontUpDown_Inpos[2]."Int"[1],
                           Bypass := #unitStatus.specialFunctions."Spare 35",
                           intOut := "Unit1.Em6.HmiInterface".intCondition.Actuator_44.intOut,
                           Moveing_INT => "Unit1.Em6.ControlNodes".cm.interlock.hotpressLeftStageLiftFront.work);
   "Unit1.Em6.ControlNodes".cmHotpressLeftStageLiftFrontUpDown.commands.commandWorkPos := NOT (NOT "Unit1.Em6.ControlNodes".hotPressLeft."step".action1[230] AND NOT "Unit1.Em6.ControlNodes".hotPressLeft."step".action1[420]) OR ((#statUnitStatus.mode.manual OR #statUnitStatus.mode.maintenance) AND "Unit1.Em6.HmiInterface".cmHotpressLeftStageLiftAllUpDown.monitoring.goToWorkPos);
END_REGION

REGION Network 38: Call CM Hot Press Left Stage Lift Front Up/Down (LBC_TwoWayActuator)
   // _."BA060ZSIBK12.10"
   RUNG wire#powerrail
      #instCmHotPressLeftStageLiftFrontUpDown(enable := TRUE, parentReferenceDesignator :=, feedbackHomePos := "BA060ZSIBK12.02", feedbackWorkPos := "BA060ZSIBK12.10", enableManualCmds := #statEnableManualCmds, interlockHomePos := "Unit1.Em6.ControlNodes".cm.interlock.hotpressLeftStageLiftFront.home, interlockWorkPos := "Unit1.Em6.ControlNodes".cm.interlock.hotpressLeftStageLiftFront.work, configuration := "Unit1.Em6.Config".cmHotpressLeftStageLiftFrontUpDown, moduleInterface := "Unit1.Em6.HmiInterface".cmHotpressLeftStageLiftFrontUpDown, controlNode := "Unit1.Em6.ControlNodes".cmHotpressLeftStageLiftFrontUpDown, goToHomePos => "BA060ZSIPM07.11", goToWorkPos => "BA060ZSIPM07.10")
   END_RUNG
   // the same network as SCL:
   #instCmHotPressLeftStageLiftFrontUpDown(enable := TRUE,   // "LBC_TwoWayActuatorCn"
                           feedbackHomePos := "BA060ZSIBK12.02",
                           feedbackWorkPos := "BA060ZSIBK12.10",
                           enableManualCmds := #statEnableManualCmds,
                           interlockHomePos := "Unit1.Em6.ControlNodes".cm.interlock.hotpressLeftStageLiftFront.home,
                           interlockWorkPos := "Unit1.Em6.ControlNodes".cm.interlock.hotpressLeftStageLiftFront.work,
                           configuration := "Unit1.Em6.Config".cmHotpressLeftStageLiftFrontUpDown,
                           moduleInterface := "Unit1.Em6.HmiInterface".cmHotpressLeftStageLiftFrontUpDown,
                           controlNode := "Unit1.Em6.ControlNodes".cmHotpressLeftStageLiftFrontUpDown,
                           goToHomePos => "BA060ZSIPM07.11",
                           goToWorkPos => "BA060ZSIPM07.10");
END_REGION

REGION Network 40: Hot Press Left Stage Lift Rear Interlock Condition
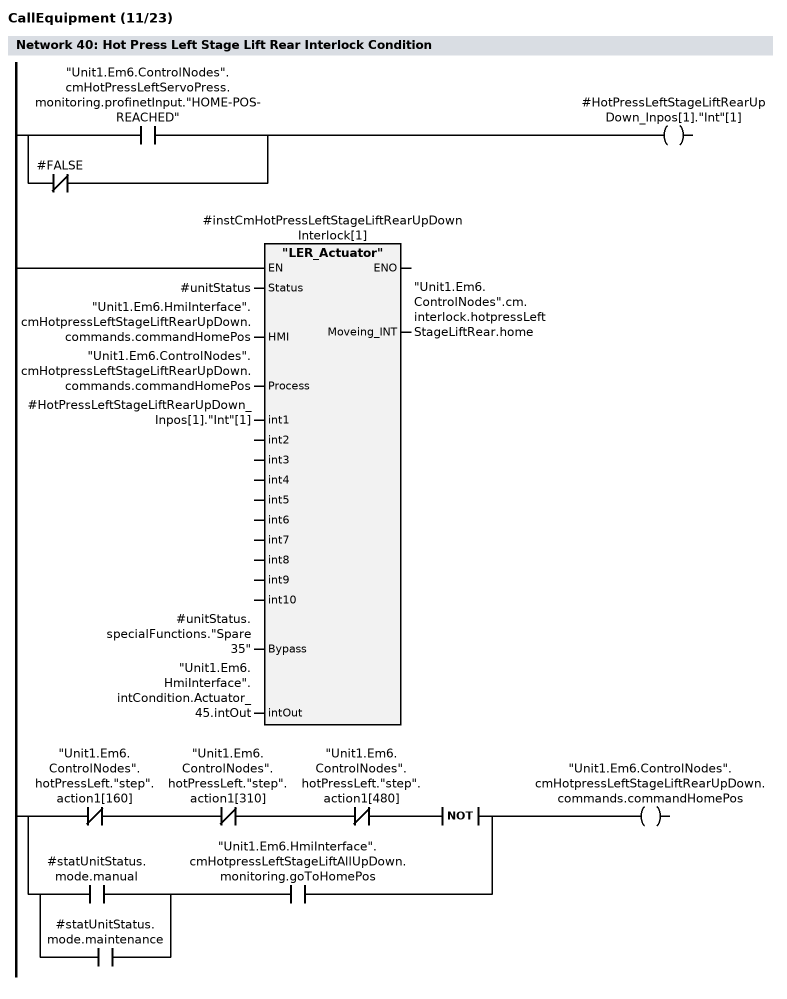
   RUNG wire#powerrail
      Contact( "Unit1.Em6.ControlNodes".cmHotPressLeftServoPress.monitoring.profinetInput."HOME-POS-REACHED" )
      wire#w1
      Coil( #HotPressLeftStageLiftRearUpDown_Inpos[1]."Int"[1] )
   END_RUNG
   RUNG wire#powerrail
      I_Contact( #FALSE )
   END_RUNG wire#w1
   RUNG wire#powerrail
      #instCmHotPressLeftStageLiftRearUpDownInterlock[1](Status := #unitStatus, HMI := "Unit1.Em6.HmiInterface".cmHotpressLeftStageLiftRearUpDown.commands.commandHomePos, Process := "Unit1.Em6.ControlNodes".cmHotpressLeftStageLiftRearUpDown.commands.commandHomePos, int1 := #HotPressLeftStageLiftRearUpDown_Inpos[1]."Int"[1], int2 :=, int3 :=, int4 :=, int5 :=, int6 :=, int7 :=, int8 :=, int9 :=, int10 :=, Bypass := #unitStatus.specialFunctions."Spare 35", intOut := "Unit1.Em6.HmiInterface".intCondition.Actuator_45.intOut, Moveing_INT => "Unit1.Em6.ControlNodes".cm.interlock.hotpressLeftStageLiftRear.home)
   END_RUNG
   RUNG wire#powerrail
      I_Contact( "Unit1.Em6.ControlNodes".hotPressLeft."step".action1[160] )
      I_Contact( "Unit1.Em6.ControlNodes".hotPressLeft."step".action1[310] )
      I_Contact( "Unit1.Em6.ControlNodes".hotPressLeft."step".action1[480] )
      Not()
      wire#w2
      Coil( "Unit1.Em6.ControlNodes".cmHotpressLeftStageLiftRearUpDown.commands.commandHomePos )
   END_RUNG
   RUNG wire#powerrail
      Contact( #statUnitStatus.mode.manual )
      wire#w3
      Contact( "Unit1.Em6.HmiInterface".cmHotpressLeftStageLiftAllUpDown.monitoring.goToHomePos )
   END_RUNG wire#w2
   RUNG wire#powerrail
      Contact( #statUnitStatus.mode.maintenance )
   END_RUNG wire#w3
   // the same network as SCL:
   #HotPressLeftStageLiftRearUpDown_Inpos[1]."Int"[1] := "Unit1.Em6.ControlNodes".cmHotPressLeftServoPress.monitoring.profinetInput."HOME-POS-REACHED" OR NOT #FALSE;
   #instCmHotPressLeftStageLiftRearUpDownInterlock[1](Status := #unitStatus,   // "LER_Actuator"
                           HMI := "Unit1.Em6.HmiInterface".cmHotpressLeftStageLiftRearUpDown.commands.commandHomePos,
                           Process := "Unit1.Em6.ControlNodes".cmHotpressLeftStageLiftRearUpDown.commands.commandHomePos,
                           int1 := #HotPressLeftStageLiftRearUpDown_Inpos[1]."Int"[1],
                           Bypass := #unitStatus.specialFunctions."Spare 35",
                           intOut := "Unit1.Em6.HmiInterface".intCondition.Actuator_45.intOut,
                           Moveing_INT => "Unit1.Em6.ControlNodes".cm.interlock.hotpressLeftStageLiftRear.home);
   "Unit1.Em6.ControlNodes".cmHotpressLeftStageLiftRearUpDown.commands.commandHomePos := NOT (NOT "Unit1.Em6.ControlNodes".hotPressLeft."step".action1[160] AND NOT "Unit1.Em6.ControlNodes".hotPressLeft."step".action1[310] AND NOT "Unit1.Em6.ControlNodes".hotPressLeft."step".action1[480]) OR ((#statUnitStatus.mode.manual OR #statUnitStatus.mode.maintenance) AND "Unit1.Em6.HmiInterface".cmHotpressLeftStageLiftAllUpDown.monitoring.goToHomePos);
END_REGION

REGION Network 41: Hot Press Left Stage Lift Rear Commands
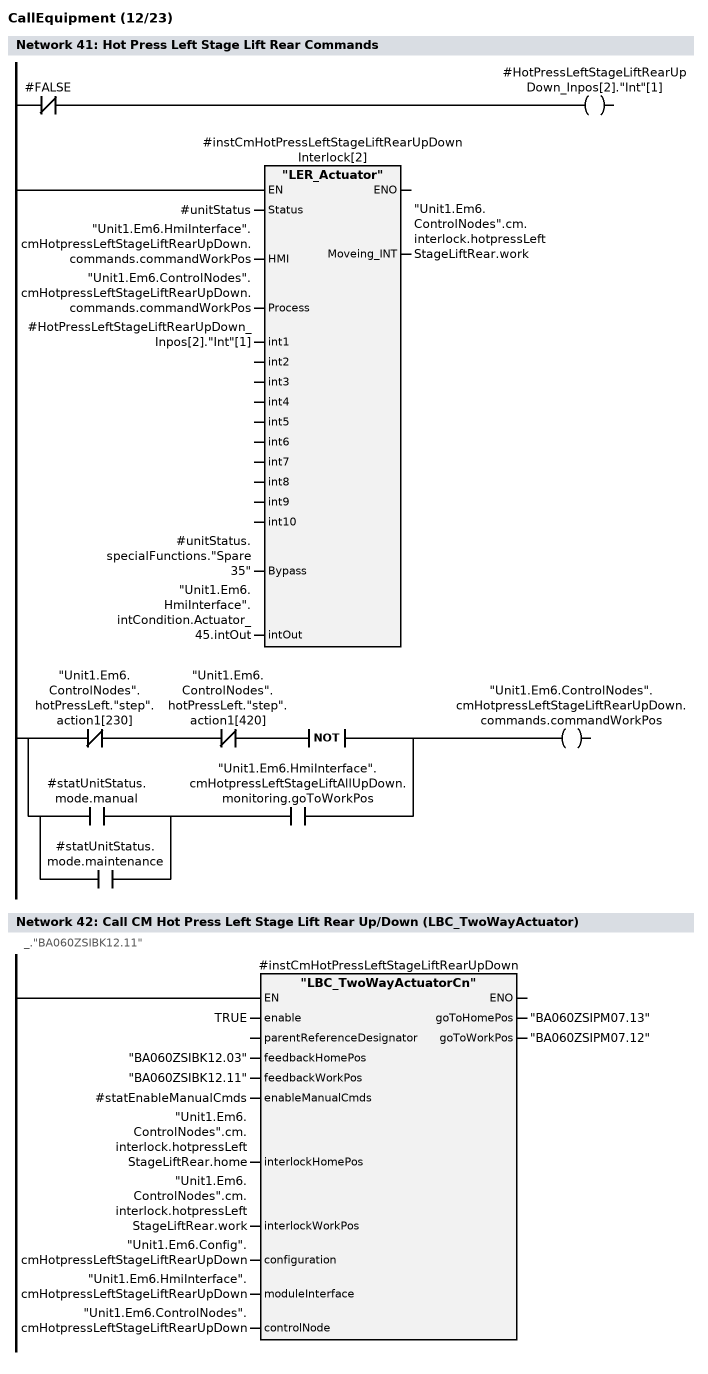
   RUNG wire#powerrail
      I_Contact( #FALSE )
      Coil( #HotPressLeftStageLiftRearUpDown_Inpos[2]."Int"[1] )
   END_RUNG
   RUNG wire#powerrail
      #instCmHotPressLeftStageLiftRearUpDownInterlock[2](Status := #unitStatus, HMI := "Unit1.Em6.HmiInterface".cmHotpressLeftStageLiftRearUpDown.commands.commandWorkPos, Process := "Unit1.Em6.ControlNodes".cmHotpressLeftStageLiftRearUpDown.commands.commandWorkPos, int1 := #HotPressLeftStageLiftRearUpDown_Inpos[2]."Int"[1], int2 :=, int3 :=, int4 :=, int5 :=, int6 :=, int7 :=, int8 :=, int9 :=, int10 :=, Bypass := #unitStatus.specialFunctions."Spare 35", intOut := "Unit1.Em6.HmiInterface".intCondition.Actuator_45.intOut, Moveing_INT => "Unit1.Em6.ControlNodes".cm.interlock.hotpressLeftStageLiftRear.work)
   END_RUNG
   RUNG wire#powerrail
      I_Contact( "Unit1.Em6.ControlNodes".hotPressLeft."step".action1[230] )
      I_Contact( "Unit1.Em6.ControlNodes".hotPressLeft."step".action1[420] )
      Not()
      wire#w1
      Coil( "Unit1.Em6.ControlNodes".cmHotpressLeftStageLiftRearUpDown.commands.commandWorkPos )
   END_RUNG
   RUNG wire#powerrail
      Contact( #statUnitStatus.mode.manual )
      wire#w2
      Contact( "Unit1.Em6.HmiInterface".cmHotpressLeftStageLiftAllUpDown.monitoring.goToWorkPos )
   END_RUNG wire#w1
   RUNG wire#powerrail
      Contact( #statUnitStatus.mode.maintenance )
   END_RUNG wire#w2
   // the same network as SCL:
   #HotPressLeftStageLiftRearUpDown_Inpos[2]."Int"[1] := NOT #FALSE;
   #instCmHotPressLeftStageLiftRearUpDownInterlock[2](Status := #unitStatus,   // "LER_Actuator"
                           HMI := "Unit1.Em6.HmiInterface".cmHotpressLeftStageLiftRearUpDown.commands.commandWorkPos,
                           Process := "Unit1.Em6.ControlNodes".cmHotpressLeftStageLiftRearUpDown.commands.commandWorkPos,
                           int1 := #HotPressLeftStageLiftRearUpDown_Inpos[2]."Int"[1],
                           Bypass := #unitStatus.specialFunctions."Spare 35",
                           intOut := "Unit1.Em6.HmiInterface".intCondition.Actuator_45.intOut,
                           Moveing_INT => "Unit1.Em6.ControlNodes".cm.interlock.hotpressLeftStageLiftRear.work);
   "Unit1.Em6.ControlNodes".cmHotpressLeftStageLiftRearUpDown.commands.commandWorkPos := NOT (NOT "Unit1.Em6.ControlNodes".hotPressLeft."step".action1[230] AND NOT "Unit1.Em6.ControlNodes".hotPressLeft."step".action1[420]) OR ((#statUnitStatus.mode.manual OR #statUnitStatus.mode.maintenance) AND "Unit1.Em6.HmiInterface".cmHotpressLeftStageLiftAllUpDown.monitoring.goToWorkPos);
END_REGION

REGION Network 42: Call CM Hot Press Left Stage Lift Rear Up/Down (LBC_TwoWayActuator)
   // _."BA060ZSIBK12.11"
   RUNG wire#powerrail
      #instCmHotPressLeftStageLiftRearUpDown(enable := TRUE, parentReferenceDesignator :=, feedbackHomePos := "BA060ZSIBK12.03", feedbackWorkPos := "BA060ZSIBK12.11", enableManualCmds := #statEnableManualCmds, interlockHomePos := "Unit1.Em6.ControlNodes".cm.interlock.hotpressLeftStageLiftRear.home, interlockWorkPos := "Unit1.Em6.ControlNodes".cm.interlock.hotpressLeftStageLiftRear.work, configuration := "Unit1.Em6.Config".cmHotpressLeftStageLiftRearUpDown, moduleInterface := "Unit1.Em6.HmiInterface".cmHotpressLeftStageLiftRearUpDown, controlNode := "Unit1.Em6.ControlNodes".cmHotpressLeftStageLiftRearUpDown, goToHomePos => "BA060ZSIPM07.13", goToWorkPos => "BA060ZSIPM07.12")
   END_RUNG
   // the same network as SCL:
   #instCmHotPressLeftStageLiftRearUpDown(enable := TRUE,   // "LBC_TwoWayActuatorCn"
                           feedbackHomePos := "BA060ZSIBK12.03",
                           feedbackWorkPos := "BA060ZSIBK12.11",
                           enableManualCmds := #statEnableManualCmds,
                           interlockHomePos := "Unit1.Em6.ControlNodes".cm.interlock.hotpressLeftStageLiftRear.home,
                           interlockWorkPos := "Unit1.Em6.ControlNodes".cm.interlock.hotpressLeftStageLiftRear.work,
                           configuration := "Unit1.Em6.Config".cmHotpressLeftStageLiftRearUpDown,
                           moduleInterface := "Unit1.Em6.HmiInterface".cmHotpressLeftStageLiftRearUpDown,
                           controlNode := "Unit1.Em6.ControlNodes".cmHotpressLeftStageLiftRearUpDown,
                           goToHomePos => "BA060ZSIPM07.13",
                           goToWorkPos => "BA060ZSIPM07.12");
END_REGION

REGION Network 44: Hot Press Left Stage Lift All Interlock Condition
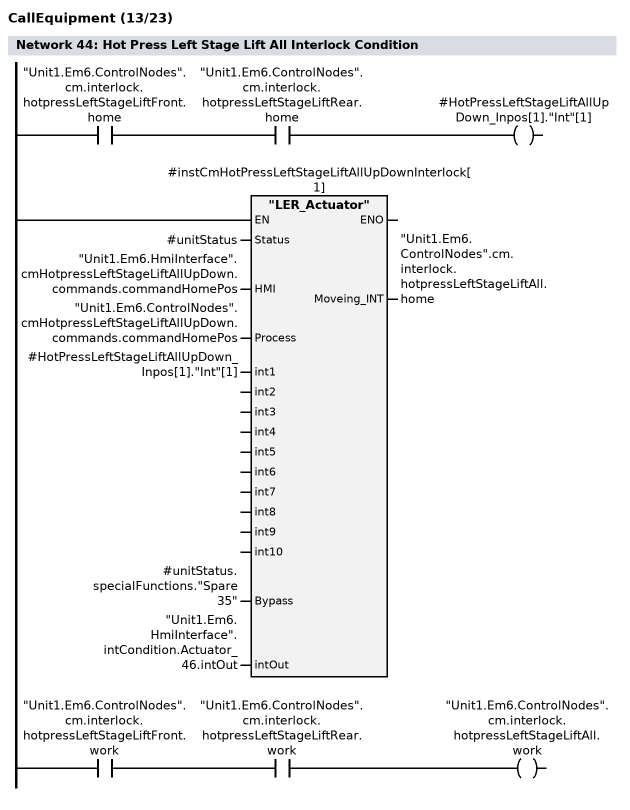
   RUNG wire#powerrail
      Contact( "Unit1.Em6.ControlNodes".cm.interlock.hotpressLeftStageLiftFront.home )
      Contact( "Unit1.Em6.ControlNodes".cm.interlock.hotpressLeftStageLiftRear.home )
      Coil( #HotPressLeftStageLiftAllUpDown_Inpos[1]."Int"[1] )
   END_RUNG
   RUNG wire#powerrail
      #instCmHotPressLeftStageLiftAllUpDownInterlock[1](Status := #unitStatus, HMI := "Unit1.Em6.HmiInterface".cmHotpressLeftStageLiftAllUpDown.commands.commandHomePos, Process := "Unit1.Em6.ControlNodes".cmHotpressLeftStageLiftAllUpDown.commands.commandHomePos, int1 := #HotPressLeftStageLiftAllUpDown_Inpos[1]."Int"[1], int2 :=, int3 :=, int4 :=, int5 :=, int6 :=, int7 :=, int8 :=, int9 :=, int10 :=, Bypass := #unitStatus.specialFunctions."Spare 35", intOut := "Unit1.Em6.HmiInterface".intCondition.Actuator_46.intOut, Moveing_INT => "Unit1.Em6.ControlNodes".cm.interlock.hotpressLeftStageLiftAll.home)
   END_RUNG
   RUNG wire#powerrail
      Contact( "Unit1.Em6.ControlNodes".cm.interlock.hotpressLeftStageLiftFront.work )
      Contact( "Unit1.Em6.ControlNodes".cm.interlock.hotpressLeftStageLiftRear.work )
      Coil( "Unit1.Em6.ControlNodes".cm.interlock.hotpressLeftStageLiftAll.work )
   END_RUNG
   // the same network as SCL:
   #HotPressLeftStageLiftAllUpDown_Inpos[1]."Int"[1] := "Unit1.Em6.ControlNodes".cm.interlock.hotpressLeftStageLiftFront.home AND "Unit1.Em6.ControlNodes".cm.interlock.hotpressLeftStageLiftRear.home;
   #instCmHotPressLeftStageLiftAllUpDownInterlock[1](Status := #unitStatus,   // "LER_Actuator"
                           HMI := "Unit1.Em6.HmiInterface".cmHotpressLeftStageLiftAllUpDown.commands.commandHomePos,
                           Process := "Unit1.Em6.ControlNodes".cmHotpressLeftStageLiftAllUpDown.commands.commandHomePos,
                           int1 := #HotPressLeftStageLiftAllUpDown_Inpos[1]."Int"[1],
                           Bypass := #unitStatus.specialFunctions."Spare 35",
                           intOut := "Unit1.Em6.HmiInterface".intCondition.Actuator_46.intOut,
                           Moveing_INT => "Unit1.Em6.ControlNodes".cm.interlock.hotpressLeftStageLiftAll.home);
   "Unit1.Em6.ControlNodes".cm.interlock.hotpressLeftStageLiftAll.work := "Unit1.Em6.ControlNodes".cm.interlock.hotpressLeftStageLiftFront.work AND "Unit1.Em6.ControlNodes".cm.interlock.hotpressLeftStageLiftRear.work;
END_REGION

REGION Network 45: Hot Press Left Stage Lift All Interlock Condition
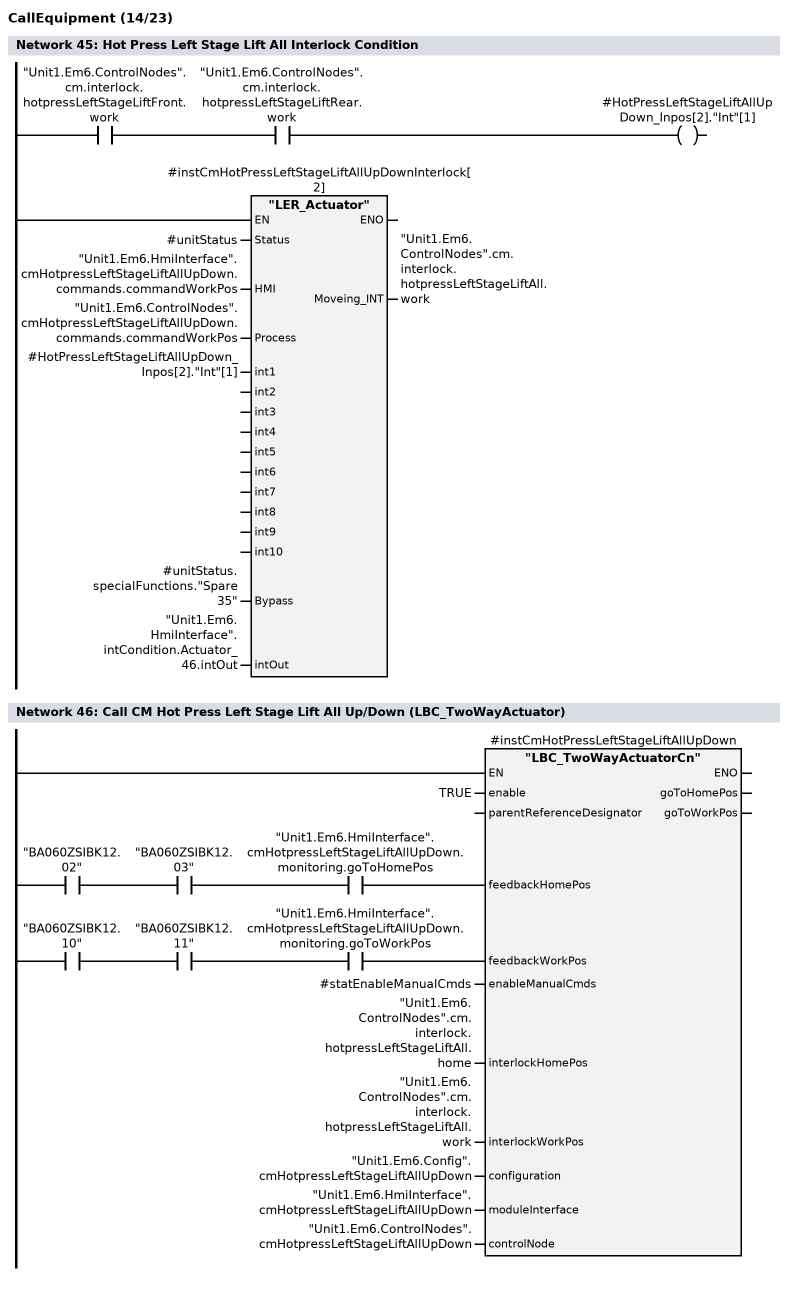
   RUNG wire#powerrail
      Contact( "Unit1.Em6.ControlNodes".cm.interlock.hotpressLeftStageLiftFront.work )
      Contact( "Unit1.Em6.ControlNodes".cm.interlock.hotpressLeftStageLiftRear.work )
      Coil( #HotPressLeftStageLiftAllUpDown_Inpos[2]."Int"[1] )
   END_RUNG
   RUNG wire#powerrail
      #instCmHotPressLeftStageLiftAllUpDownInterlock[2](Status := #unitStatus, HMI := "Unit1.Em6.HmiInterface".cmHotpressLeftStageLiftAllUpDown.commands.commandWorkPos, Process := "Unit1.Em6.ControlNodes".cmHotpressLeftStageLiftAllUpDown.commands.commandWorkPos, int1 := #HotPressLeftStageLiftAllUpDown_Inpos[2]."Int"[1], int2 :=, int3 :=, int4 :=, int5 :=, int6 :=, int7 :=, int8 :=, int9 :=, int10 :=, Bypass := #unitStatus.specialFunctions."Spare 35", intOut := "Unit1.Em6.HmiInterface".intCondition.Actuator_46.intOut, Moveing_INT => "Unit1.Em6.ControlNodes".cm.interlock.hotpressLeftStageLiftAll.work)
   END_RUNG
   // the same network as SCL:
   #HotPressLeftStageLiftAllUpDown_Inpos[2]."Int"[1] := "Unit1.Em6.ControlNodes".cm.interlock.hotpressLeftStageLiftFront.work AND "Unit1.Em6.ControlNodes".cm.interlock.hotpressLeftStageLiftRear.work;
   #instCmHotPressLeftStageLiftAllUpDownInterlock[2](Status := #unitStatus,   // "LER_Actuator"
                           HMI := "Unit1.Em6.HmiInterface".cmHotpressLeftStageLiftAllUpDown.commands.commandWorkPos,
                           Process := "Unit1.Em6.ControlNodes".cmHotpressLeftStageLiftAllUpDown.commands.commandWorkPos,
                           int1 := #HotPressLeftStageLiftAllUpDown_Inpos[2]."Int"[1],
                           Bypass := #unitStatus.specialFunctions."Spare 35",
                           intOut := "Unit1.Em6.HmiInterface".intCondition.Actuator_46.intOut,
                           Moveing_INT => "Unit1.Em6.ControlNodes".cm.interlock.hotpressLeftStageLiftAll.work);
END_REGION

REGION Network 46: Call CM Hot Press Left Stage Lift All Up/Down (LBC_TwoWayActuator)
   RUNG wire#powerrail
      #instCmHotPressLeftStageLiftAllUpDown(feedbackHomePos := wire#w1, feedbackWorkPos := wire#w2, enable := TRUE, parentReferenceDesignator :=, enableManualCmds := #statEnableManualCmds, interlockHomePos := "Unit1.Em6.ControlNodes".cm.interlock.hotpressLeftStageLiftAll.home, interlockWorkPos := "Unit1.Em6.ControlNodes".cm.interlock.hotpressLeftStageLiftAll.work, configuration := "Unit1.Em6.Config".cmHotpressLeftStageLiftAllUpDown, moduleInterface := "Unit1.Em6.HmiInterface".cmHotpressLeftStageLiftAllUpDown, controlNode := "Unit1.Em6.ControlNodes".cmHotpressLeftStageLiftAllUpDown, goToHomePos =>, goToWorkPos =>)
   END_RUNG
   RUNG wire#powerrail
      Contact( "BA060ZSIBK12.02" )
      Contact( "BA060ZSIBK12.03" )
      Contact( "Unit1.Em6.HmiInterface".cmHotpressLeftStageLiftAllUpDown.monitoring.goToHomePos )
   END_RUNG wire#w1
   RUNG wire#powerrail
      Contact( "BA060ZSIBK12.10" )
      Contact( "BA060ZSIBK12.11" )
      Contact( "Unit1.Em6.HmiInterface".cmHotpressLeftStageLiftAllUpDown.monitoring.goToWorkPos )
   END_RUNG wire#w2
   // the same network as SCL:
   #instCmHotPressLeftStageLiftAllUpDown(enable := TRUE,   // "LBC_TwoWayActuatorCn"
                           feedbackHomePos := "BA060ZSIBK12.02" AND "BA060ZSIBK12.03" AND "Unit1.Em6.HmiInterface".cmHotpressLeftStageLiftAllUpDown.monitoring.goToHomePos,
                           feedbackWorkPos := "BA060ZSIBK12.10" AND "BA060ZSIBK12.11" AND "Unit1.Em6.HmiInterface".cmHotpressLeftStageLiftAllUpDown.monitoring.goToWorkPos,
                           enableManualCmds := #statEnableManualCmds,
                           interlockHomePos := "Unit1.Em6.ControlNodes".cm.interlock.hotpressLeftStageLiftAll.home,
                           interlockWorkPos := "Unit1.Em6.ControlNodes".cm.interlock.hotpressLeftStageLiftAll.work,
                           configuration := "Unit1.Em6.Config".cmHotpressLeftStageLiftAllUpDown,
                           moduleInterface := "Unit1.Em6.HmiInterface".cmHotpressLeftStageLiftAllUpDown,
                           controlNode := "Unit1.Em6.ControlNodes".cmHotpressLeftStageLiftAllUpDown);
END_REGION

REGION Network 48: ******************** Control Modules (Accessories) ********************
END_REGION

REGION Network 49: Temperature Limit Convert
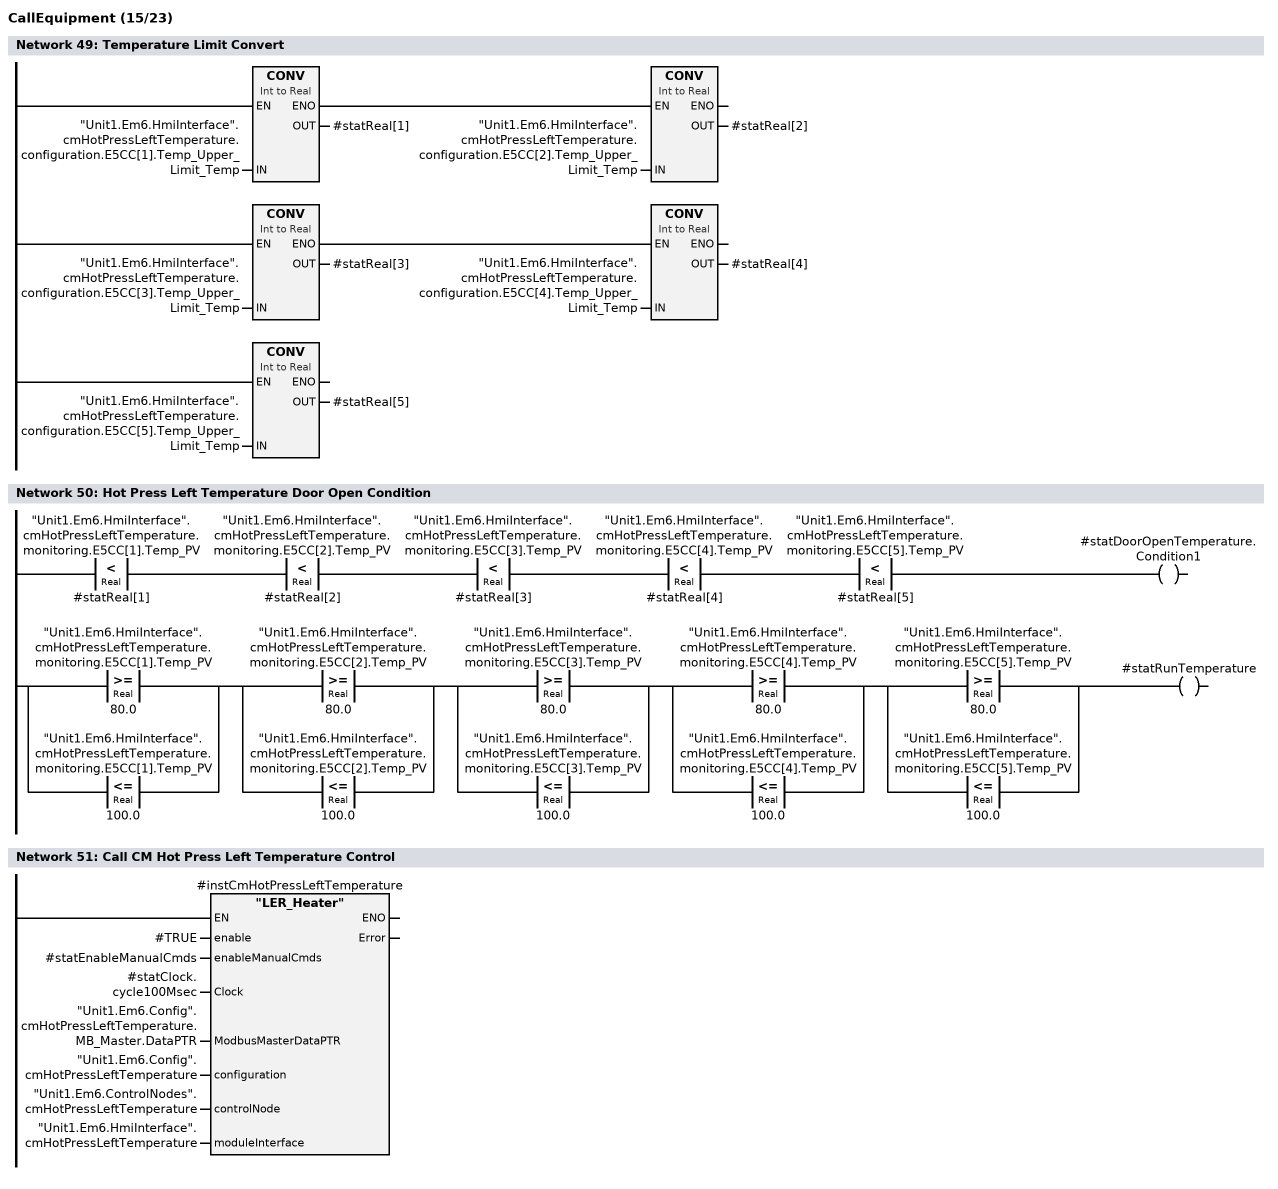
   RUNG wire#powerrail
      { S7_Templates := "[SrcType := Int, DestType := Real]" } Convert(in := "Unit1.Em6.HmiInterface".cmHotPressLeftTemperature.configuration.E5CC[1].Temp_Upper_Limit_Temp, out => #statReal[1])
      { S7_Templates := "[SrcType := Int, DestType := Real]" } Convert(in := "Unit1.Em6.HmiInterface".cmHotPressLeftTemperature.configuration.E5CC[2].Temp_Upper_Limit_Temp, out => #statReal[2])
   END_RUNG
   RUNG wire#powerrail
      { S7_Templates := "[SrcType := Int, DestType := Real]" } Convert(in := "Unit1.Em6.HmiInterface".cmHotPressLeftTemperature.configuration.E5CC[3].Temp_Upper_Limit_Temp, out => #statReal[3])
      { S7_Templates := "[SrcType := Int, DestType := Real]" } Convert(in := "Unit1.Em6.HmiInterface".cmHotPressLeftTemperature.configuration.E5CC[4].Temp_Upper_Limit_Temp, out => #statReal[4])
   END_RUNG
   RUNG wire#powerrail
      { S7_Templates := "[SrcType := Int, DestType := Real]" } Convert(in := "Unit1.Em6.HmiInterface".cmHotPressLeftTemperature.configuration.E5CC[5].Temp_Upper_Limit_Temp, out => #statReal[5])
   END_RUNG
   // the same network as SCL:
   #statReal[1] := INT_TO_REAL("Unit1.Em6.HmiInterface".cmHotPressLeftTemperature.configuration.E5CC[1].Temp_Upper_Limit_Temp);
   #statReal[2] := INT_TO_REAL("Unit1.Em6.HmiInterface".cmHotPressLeftTemperature.configuration.E5CC[2].Temp_Upper_Limit_Temp);
   #statReal[3] := INT_TO_REAL("Unit1.Em6.HmiInterface".cmHotPressLeftTemperature.configuration.E5CC[3].Temp_Upper_Limit_Temp);
   #statReal[4] := INT_TO_REAL("Unit1.Em6.HmiInterface".cmHotPressLeftTemperature.configuration.E5CC[4].Temp_Upper_Limit_Temp);
   #statReal[5] := INT_TO_REAL("Unit1.Em6.HmiInterface".cmHotPressLeftTemperature.configuration.E5CC[5].Temp_Upper_Limit_Temp);
END_REGION

REGION Network 50: Hot Press Left Temperature Door Open Condition
   RUNG wire#powerrail
      { S7_Templates := "SrcType := Real" } LT_Contact(in1 := "Unit1.Em6.HmiInterface".cmHotPressLeftTemperature.monitoring.E5CC[1].Temp_PV, in2 := #statReal[1])
      { S7_Templates := "SrcType := Real" } LT_Contact(in1 := "Unit1.Em6.HmiInterface".cmHotPressLeftTemperature.monitoring.E5CC[2].Temp_PV, in2 := #statReal[2])
      { S7_Templates := "SrcType := Real" } LT_Contact(in1 := "Unit1.Em6.HmiInterface".cmHotPressLeftTemperature.monitoring.E5CC[3].Temp_PV, in2 := #statReal[3])
      { S7_Templates := "SrcType := Real" } LT_Contact(in1 := "Unit1.Em6.HmiInterface".cmHotPressLeftTemperature.monitoring.E5CC[4].Temp_PV, in2 := #statReal[4])
      { S7_Templates := "SrcType := Real" } LT_Contact(in1 := "Unit1.Em6.HmiInterface".cmHotPressLeftTemperature.monitoring.E5CC[5].Temp_PV, in2 := #statReal[5])
      Coil( #statDoorOpenTemperature.Condition1 )
   END_RUNG
   RUNG wire#powerrail
      { S7_Templates := "SrcType := Real" } GE_Contact(in1 := "Unit1.Em6.HmiInterface".cmHotPressLeftTemperature.monitoring.E5CC[1].Temp_PV, in2 := 80.0)
      wire#w1
      { S7_Templates := "SrcType := Real" } GE_Contact(in1 := "Unit1.Em6.HmiInterface".cmHotPressLeftTemperature.monitoring.E5CC[2].Temp_PV, in2 := 80.0)
      wire#w2
      { S7_Templates := "SrcType := Real" } GE_Contact(in1 := "Unit1.Em6.HmiInterface".cmHotPressLeftTemperature.monitoring.E5CC[3].Temp_PV, in2 := 80.0)
      wire#w3
      { S7_Templates := "SrcType := Real" } GE_Contact(in1 := "Unit1.Em6.HmiInterface".cmHotPressLeftTemperature.monitoring.E5CC[4].Temp_PV, in2 := 80.0)
      wire#w4
      { S7_Templates := "SrcType := Real" } GE_Contact(in1 := "Unit1.Em6.HmiInterface".cmHotPressLeftTemperature.monitoring.E5CC[5].Temp_PV, in2 := 80.0)
      wire#w5
      Coil( #statRunTemperature )
   END_RUNG
   RUNG wire#powerrail
      { S7_Templates := "SrcType := Real" } LE_Contact(in1 := "Unit1.Em6.HmiInterface".cmHotPressLeftTemperature.monitoring.E5CC[1].Temp_PV, in2 := 100.0)
   END_RUNG wire#w1
   RUNG wire#w1
      { S7_Templates := "SrcType := Real" } LE_Contact(in1 := "Unit1.Em6.HmiInterface".cmHotPressLeftTemperature.monitoring.E5CC[2].Temp_PV, in2 := 100.0)
   END_RUNG wire#w2
   RUNG wire#w2
      { S7_Templates := "SrcType := Real" } LE_Contact(in1 := "Unit1.Em6.HmiInterface".cmHotPressLeftTemperature.monitoring.E5CC[3].Temp_PV, in2 := 100.0)
   END_RUNG wire#w3
   RUNG wire#w3
      { S7_Templates := "SrcType := Real" } LE_Contact(in1 := "Unit1.Em6.HmiInterface".cmHotPressLeftTemperature.monitoring.E5CC[4].Temp_PV, in2 := 100.0)
   END_RUNG wire#w4
   RUNG wire#w4
      { S7_Templates := "SrcType := Real" } LE_Contact(in1 := "Unit1.Em6.HmiInterface".cmHotPressLeftTemperature.monitoring.E5CC[5].Temp_PV, in2 := 100.0)
   END_RUNG wire#w5
   // the same network as SCL:
   #statDoorOpenTemperature.Condition1 := ("Unit1.Em6.HmiInterface".cmHotPressLeftTemperature.monitoring.E5CC[1].Temp_PV < #statReal[1]) AND ("Unit1.Em6.HmiInterface".cmHotPressLeftTemperature.monitoring.E5CC[2].Temp_PV < #statReal[2]) AND ("Unit1.Em6.HmiInterface".cmHotPressLeftTemperature.monitoring.E5CC[3].Temp_PV < #statReal[3]) AND ("Unit1.Em6.HmiInterface".cmHotPressLeftTemperature.monitoring.E5CC[4].Temp_PV < #statReal[4]) AND ("Unit1.Em6.HmiInterface".cmHotPressLeftTemperature.monitoring.E5CC[5].Temp_PV < #statReal[5]);
   #statRunTemperature := (("Unit1.Em6.HmiInterface".cmHotPressLeftTemperature.monitoring.E5CC[1].Temp_PV >= 80.0) OR ("Unit1.Em6.HmiInterface".cmHotPressLeftTemperature.monitoring.E5CC[1].Temp_PV <= 100.0)) AND (("Unit1.Em6.HmiInterface".cmHotPressLeftTemperature.monitoring.E5CC[2].Temp_PV >= 80.0) OR ("Unit1.Em6.HmiInterface".cmHotPressLeftTemperature.monitoring.E5CC[2].Temp_PV <= 100.0)) AND (("Unit1.Em6.HmiInterface".cmHotPressLeftTemperature.monitoring.E5CC[3].Temp_PV >= 80.0) OR ("Unit1.Em6.HmiInterface".cmHotPressLeftTemperature.monitoring.E5CC[3].Temp_PV <= 100.0)) AND (("Unit1.Em6.HmiInterface".cmHotPressLeftTemperature.monitoring.E5CC[4].Temp_PV >= 80.0) OR ("Unit1.Em6.HmiInterface".cmHotPressLeftTemperature.monitoring.E5CC[4].Temp_PV <= 100.0)) AND (("Unit1.Em6.HmiInterface".cmHotPressLeftTemperature.monitoring.E5CC[5].Temp_PV >= 80.0) OR ("Unit1.Em6.HmiInterface".cmHotPressLeftTemperature.monitoring.E5CC[5].Temp_PV <= 100.0));
END_REGION

REGION Network 51: Call CM Hot Press Left Temperature Control
   RUNG wire#powerrail
      #instCmHotPressLeftTemperature(enable := #TRUE, enableManualCmds := #statEnableManualCmds, Clock := #statClock.cycle100Msec, ModbusMasterDataPTR := "Unit1.Em6.Config".cmHotPressLeftTemperature.MB_Master.DataPTR, configuration := "Unit1.Em6.Config".cmHotPressLeftTemperature, controlNode := "Unit1.Em6.ControlNodes".cmHotPressLeftTemperature, moduleInterface := "Unit1.Em6.HmiInterface".cmHotPressLeftTemperature, Error =>)
   END_RUNG
   // the same network as SCL:
   #instCmHotPressLeftTemperature(enable := #TRUE,   // "LER_Heater"
                           enableManualCmds := #statEnableManualCmds,
                           Clock := #statClock.cycle100Msec,
                           ModbusMasterDataPTR := "Unit1.Em6.Config".cmHotPressLeftTemperature.MB_Master.DataPTR,
                           configuration := "Unit1.Em6.Config".cmHotPressLeftTemperature,
                           controlNode := "Unit1.Em6.ControlNodes".cmHotPressLeftTemperature,
                           moduleInterface := "Unit1.Em6.HmiInterface".cmHotPressLeftTemperature);
END_REGION

REGION Network 52: Servo Press Interlock Condition
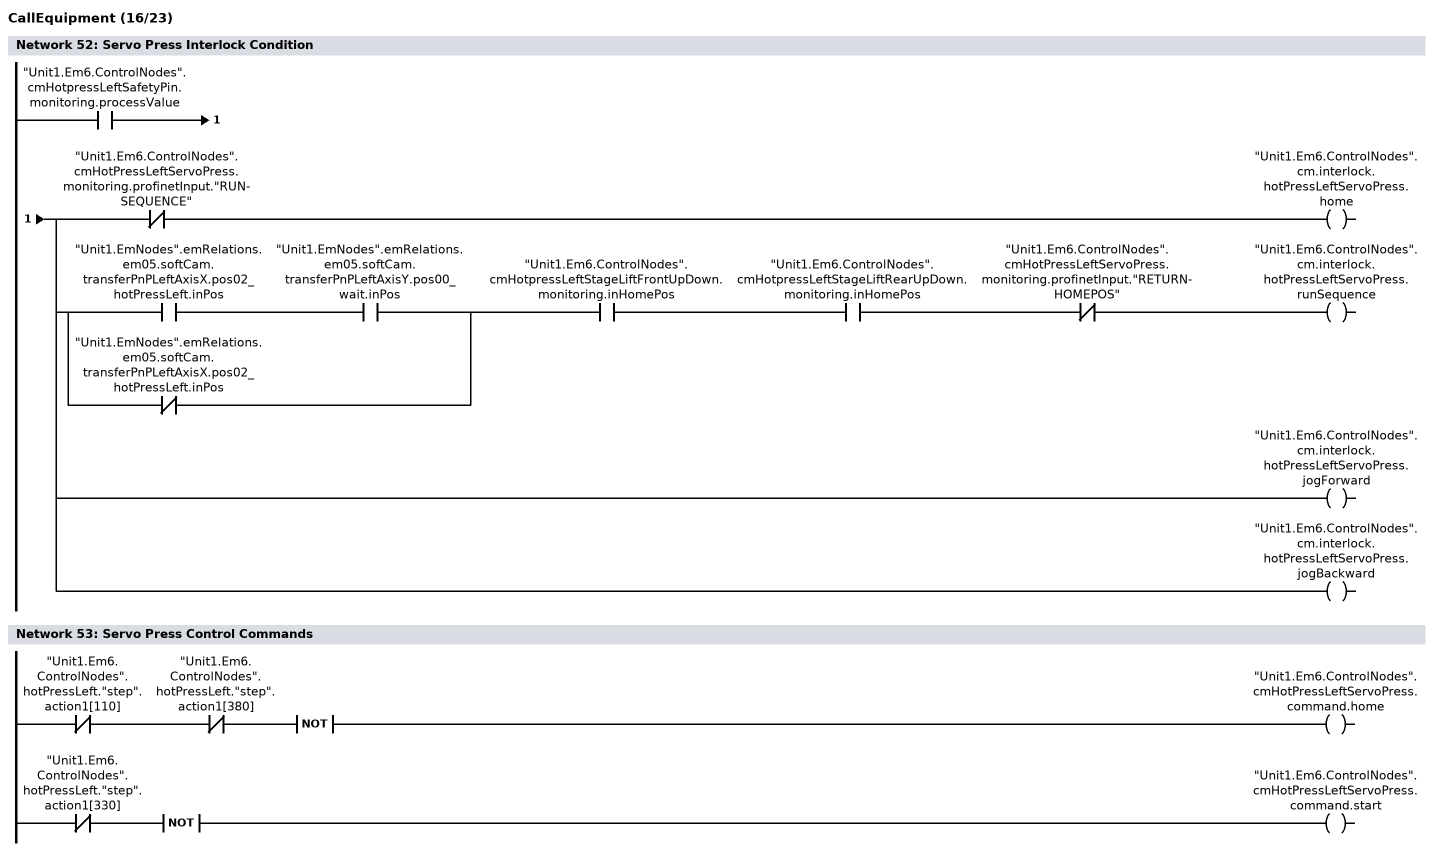
   RUNG wire#powerrail
      Contact( "Unit1.Em6.ControlNodes".cmHotpressLeftSafetyPin.monitoring.processValue )
      wire#w1
      I_Contact( "Unit1.Em6.ControlNodes".cmHotPressLeftServoPress.monitoring.profinetInput."RUN-SEQUENCE" )
      Coil( "Unit1.Em6.ControlNodes".cm.interlock.hotPressLeftServoPress.home )
   END_RUNG
   RUNG wire#w1
      Contact( "Unit1.EmNodes".emRelations.em05.softCam.transferPnPLeftAxisX.pos02_hotPressLeft.inPos )
      Contact( "Unit1.EmNodes".emRelations.em05.softCam.transferPnPLeftAxisY.pos00_wait.inPos )
      wire#w2
      Contact( "Unit1.Em6.ControlNodes".cmHotpressLeftStageLiftFrontUpDown.monitoring.inHomePos )
      Contact( "Unit1.Em6.ControlNodes".cmHotpressLeftStageLiftRearUpDown.monitoring.inHomePos )
      I_Contact( "Unit1.Em6.ControlNodes".cmHotPressLeftServoPress.monitoring.profinetInput."RETURN-HOMEPOS" )
      Coil( "Unit1.Em6.ControlNodes".cm.interlock.hotPressLeftServoPress.runSequence )
   END_RUNG
   RUNG wire#w1
      I_Contact( "Unit1.EmNodes".emRelations.em05.softCam.transferPnPLeftAxisX.pos02_hotPressLeft.inPos )
   END_RUNG wire#w2
   RUNG wire#w1
      Coil( "Unit1.Em6.ControlNodes".cm.interlock.hotPressLeftServoPress.jogForward )
   END_RUNG
   RUNG wire#w1
      Coil( "Unit1.Em6.ControlNodes".cm.interlock.hotPressLeftServoPress.jogBackward )
   END_RUNG
   // the same network as SCL:
   "Unit1.Em6.ControlNodes".cm.interlock.hotPressLeftServoPress.home := "Unit1.Em6.ControlNodes".cmHotpressLeftSafetyPin.monitoring.processValue AND NOT "Unit1.Em6.ControlNodes".cmHotPressLeftServoPress.monitoring.profinetInput."RUN-SEQUENCE";
   "Unit1.Em6.ControlNodes".cm.interlock.hotPressLeftServoPress.runSequence := "Unit1.Em6.ControlNodes".cmHotpressLeftSafetyPin.monitoring.processValue AND (("Unit1.EmNodes".emRelations.em05.softCam.transferPnPLeftAxisX.pos02_hotPressLeft.inPos AND "Unit1.EmNodes".emRelations.em05.softCam.transferPnPLeftAxisY.pos00_wait.inPos) OR NOT "Unit1.EmNodes".emRelations.em05.softCam.transferPnPLeftAxisX.pos02_hotPressLeft.inPos) AND "Unit1.Em6.ControlNodes".cmHotpressLeftStageLiftFrontUpDown.monitoring.inHomePos AND "Unit1.Em6.ControlNodes".cmHotpressLeftStageLiftRearUpDown.monitoring.inHomePos AND NOT "Unit1.Em6.ControlNodes".cmHotPressLeftServoPress.monitoring.profinetInput."RETURN-HOMEPOS";
   "Unit1.Em6.ControlNodes".cm.interlock.hotPressLeftServoPress.jogForward := "Unit1.Em6.ControlNodes".cmHotpressLeftSafetyPin.monitoring.processValue;
   "Unit1.Em6.ControlNodes".cm.interlock.hotPressLeftServoPress.jogBackward := "Unit1.Em6.ControlNodes".cmHotpressLeftSafetyPin.monitoring.processValue;
END_REGION

REGION Network 53: Servo Press Control Commands
   RUNG wire#powerrail
      I_Contact( "Unit1.Em6.ControlNodes".hotPressLeft."step".action1[110] )
      I_Contact( "Unit1.Em6.ControlNodes".hotPressLeft."step".action1[380] )
      Not()
      Coil( "Unit1.Em6.ControlNodes".cmHotPressLeftServoPress.command.home )
   END_RUNG
   RUNG wire#powerrail
      I_Contact( "Unit1.Em6.ControlNodes".hotPressLeft."step".action1[330] )
      Not()
      Coil( "Unit1.Em6.ControlNodes".cmHotPressLeftServoPress.command.start )
   END_RUNG
   // the same network as SCL:
   "Unit1.Em6.ControlNodes".cmHotPressLeftServoPress.command.home := NOT (NOT "Unit1.Em6.ControlNodes".hotPressLeft."step".action1[110] AND NOT "Unit1.Em6.ControlNodes".hotPressLeft."step".action1[380]);
   "Unit1.Em6.ControlNodes".cmHotPressLeftServoPress.command.start := NOT (NOT "Unit1.Em6.ControlNodes".hotPressLeft."step".action1[330]);
END_REGION

REGION Network 54: Call CM Servo Press Control
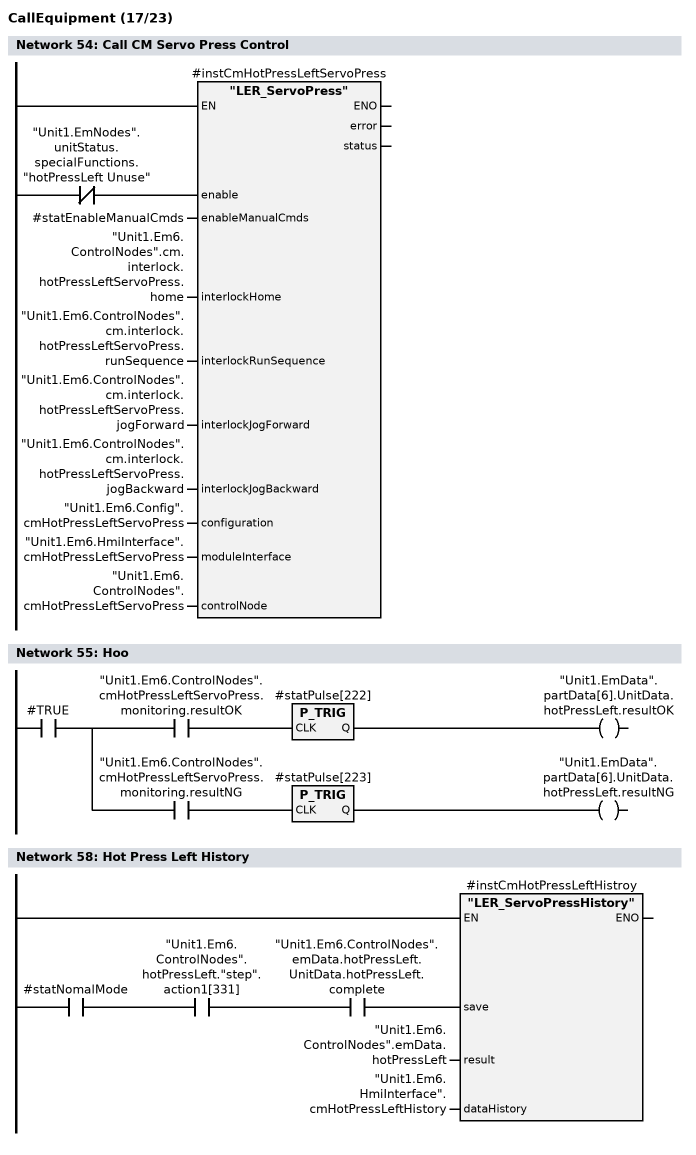
   RUNG wire#powerrail
      #instCmHotPressLeftServoPress(enable := wire#w1, enableManualCmds := #statEnableManualCmds, interlockHome := "Unit1.Em6.ControlNodes".cm.interlock.hotPressLeftServoPress.home, interlockRunSequence := "Unit1.Em6.ControlNodes".cm.interlock.hotPressLeftServoPress.runSequence, interlockJogForward := "Unit1.Em6.ControlNodes".cm.interlock.hotPressLeftServoPress.jogForward, interlockJogBackward := "Unit1.Em6.ControlNodes".cm.interlock.hotPressLeftServoPress.jogBackward, configuration := "Unit1.Em6.Config".cmHotPressLeftServoPress, moduleInterface := "Unit1.Em6.HmiInterface".cmHotPressLeftServoPress, controlNode := "Unit1.Em6.ControlNodes".cmHotPressLeftServoPress, error =>, status =>)
   END_RUNG
   RUNG wire#powerrail
      I_Contact( "Unit1.EmNodes".unitStatus.specialFunctions."hotPressLeft Unuse" )
   END_RUNG wire#w1
   // the same network as SCL:
   #instCmHotPressLeftServoPress(enable := NOT "Unit1.EmNodes".unitStatus.specialFunctions."hotPressLeft Unuse",   // "LER_ServoPress"
                           enableManualCmds := #statEnableManualCmds,
                           interlockHome := "Unit1.Em6.ControlNodes".cm.interlock.hotPressLeftServoPress.home,
                           interlockRunSequence := "Unit1.Em6.ControlNodes".cm.interlock.hotPressLeftServoPress.runSequence,
                           interlockJogForward := "Unit1.Em6.ControlNodes".cm.interlock.hotPressLeftServoPress.jogForward,
                           interlockJogBackward := "Unit1.Em6.ControlNodes".cm.interlock.hotPressLeftServoPress.jogBackward,
                           configuration := "Unit1.Em6.Config".cmHotPressLeftServoPress,
                           moduleInterface := "Unit1.Em6.HmiInterface".cmHotPressLeftServoPress,
                           controlNode := "Unit1.Em6.ControlNodes".cmHotPressLeftServoPress);
END_REGION

REGION Network 55: Hoo
   RUNG wire#powerrail
      Contact( #TRUE )
      wire#w1
      Contact( "Unit1.Em6.ControlNodes".cmHotPressLeftServoPress.monitoring.resultOK )
      P_Trig( #statPulse[222] )
      Coil( "Unit1.EmData".partData[6].UnitData.hotPressLeft.resultOK )
   END_RUNG
   RUNG wire#w1
      Contact( "Unit1.Em6.ControlNodes".cmHotPressLeftServoPress.monitoring.resultNG )
      P_Trig( #statPulse[223] )
      Coil( "Unit1.EmData".partData[6].UnitData.hotPressLeft.resultNG )
   END_RUNG
   // the same network as SCL:
   #_w1 := #TRUE AND "Unit1.Em6.ControlNodes".cmHotPressLeftServoPress.monitoring.resultOK;
   #_w2 := #_w1 AND NOT #statPulse[222];   // rising edge
   #statPulse[222] := #_w1;
   "Unit1.EmData".partData[6].UnitData.hotPressLeft.resultOK := #_w2;
   #_w3 := #TRUE AND "Unit1.Em6.ControlNodes".cmHotPressLeftServoPress.monitoring.resultNG;
   #_w4 := #_w3 AND NOT #statPulse[223];   // rising edge
   #statPulse[223] := #_w3;
   "Unit1.EmData".partData[6].UnitData.hotPressLeft.resultNG := #_w4;
END_REGION

REGION Network 57: ******************** History ********************
END_REGION

REGION Network 58: Hot Press Left History
   RUNG wire#powerrail
      #instCmHotPressLeftHistroy(save := wire#w1, result := "Unit1.Em6.ControlNodes".emData.hotPressLeft, dataHistory := "Unit1.Em6.HmiInterface".cmHotPressLeftHistory)
   END_RUNG
   RUNG wire#powerrail
      Contact( #statNomalMode )
      Contact( "Unit1.Em6.ControlNodes".hotPressLeft."step".action1[331] )
      Contact( "Unit1.Em6.ControlNodes".emData.hotPressLeft.UnitData.hotPressLeft.complete )
   END_RUNG wire#w1
   // the same network as SCL:
   #instCmHotPressLeftHistroy(save := #statNomalMode AND "Unit1.Em6.ControlNodes".hotPressLeft."step".action1[331] AND "Unit1.Em6.ControlNodes".emData.hotPressLeft.UnitData.hotPressLeft.complete,   // "LER_ServoPressHistory"
                           result := "Unit1.Em6.ControlNodes".emData.hotPressLeft,
                           dataHistory := "Unit1.Em6.HmiInterface".cmHotPressLeftHistory);
END_REGION

REGION Network 60: ******************** Feedback to Unit ********************
END_REGION

REGION Network 61: Determine StateComplete (SC) in Mode Production
   // Conditions for the Equipment Modules "stateComplete" feedback to the unit. This feedback is given when the task in for the respective state is complete.
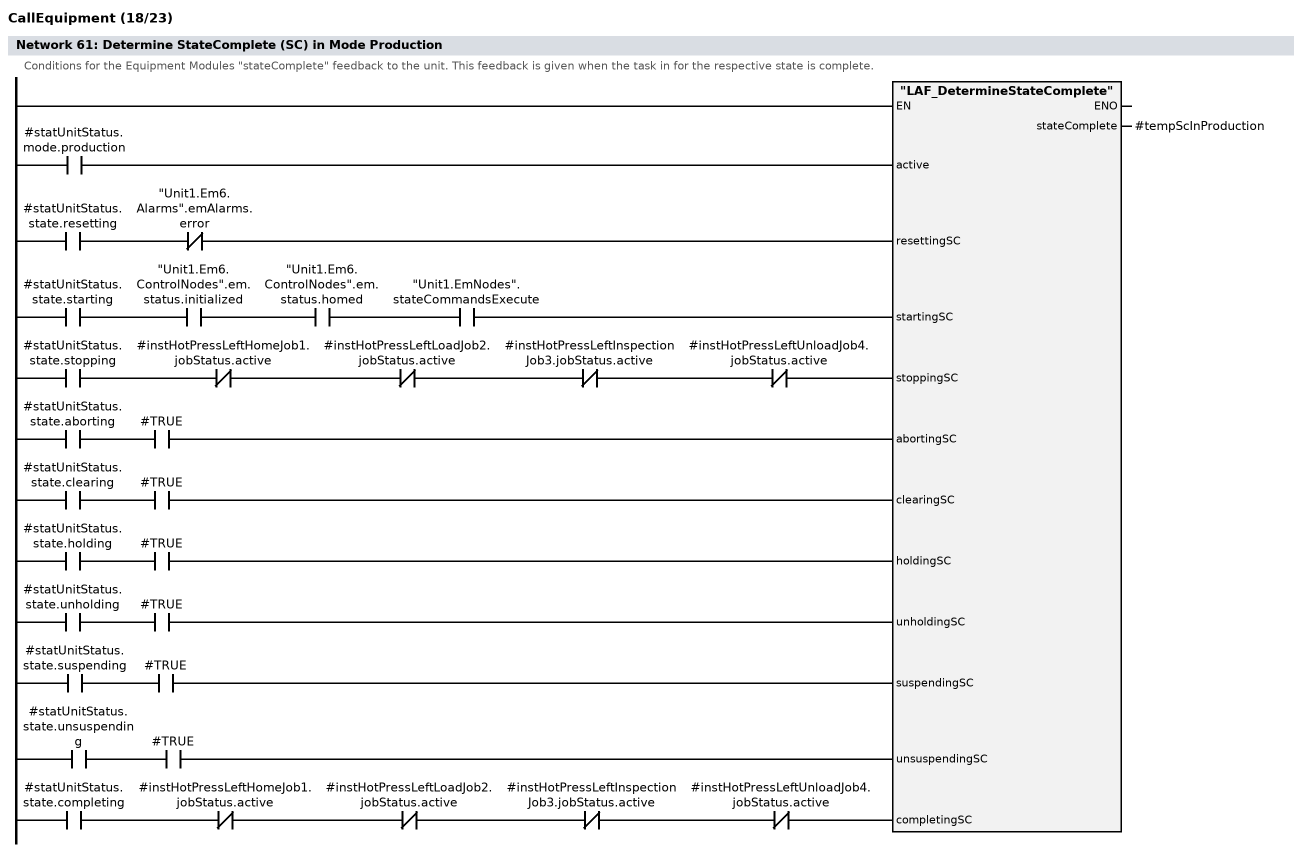
   RUNG wire#powerrail
      "LAF_DetermineStateComplete"(active := wire#w1, resettingSC := wire#w2, startingSC := wire#w3, stoppingSC := wire#w4, abortingSC := wire#w5, clearingSC := wire#w6, holdingSC := wire#w7, unholdingSC := wire#w8, suspendingSC := wire#w9, unsuspendingSC := wire#w10, completingSC := wire#w11, stateComplete => #tempScInProduction)
   END_RUNG
   RUNG wire#powerrail
      Contact( #statUnitStatus.mode.production )
   END_RUNG wire#w1
   RUNG wire#powerrail
      Contact( #statUnitStatus.state.resetting )
      I_Contact( "Unit1.Em6.Alarms".emAlarms.error )
   END_RUNG wire#w2
   RUNG wire#powerrail
      Contact( #statUnitStatus.state.starting )
      Contact( "Unit1.Em6.ControlNodes".em.status.initialized )
      Contact( "Unit1.Em6.ControlNodes".em.status.homed )
      Contact( "Unit1.EmNodes".stateCommandsExecute )
   END_RUNG wire#w3
   RUNG wire#powerrail
      Contact( #statUnitStatus.state.stopping )
      I_Contact( #instHotPressLeftHomeJob1.jobStatus.active )
      I_Contact( #instHotPressLeftLoadJob2.jobStatus.active )
      I_Contact( #instHotPressLeftInspectionJob3.jobStatus.active )
      I_Contact( #instHotPressLeftUnloadJob4.jobStatus.active )
   END_RUNG wire#w4
   RUNG wire#powerrail
      Contact( #statUnitStatus.state.aborting )
      Contact( #TRUE )
   END_RUNG wire#w5
   RUNG wire#powerrail
      Contact( #statUnitStatus.state.clearing )
      Contact( #TRUE )
   END_RUNG wire#w6
   RUNG wire#powerrail
      Contact( #statUnitStatus.state.holding )
      Contact( #TRUE )
   END_RUNG wire#w7
   RUNG wire#powerrail
      Contact( #statUnitStatus.state.unholding )
      Contact( #TRUE )
   END_RUNG wire#w8
   RUNG wire#powerrail
      Contact( #statUnitStatus.state.suspending )
      Contact( #TRUE )
   END_RUNG wire#w9
   RUNG wire#powerrail
      Contact( #statUnitStatus.state.unsuspending )
      Contact( #TRUE )
   END_RUNG wire#w10
   RUNG wire#powerrail
      Contact( #statUnitStatus.state.completing )
      I_Contact( #instHotPressLeftHomeJob1.jobStatus.active )
      I_Contact( #instHotPressLeftLoadJob2.jobStatus.active )
      I_Contact( #instHotPressLeftInspectionJob3.jobStatus.active )
      I_Contact( #instHotPressLeftUnloadJob4.jobStatus.active )
   END_RUNG wire#w11
   // the same network as SCL:
   "LAF_DetermineStateComplete"(active := #statUnitStatus.mode.production,
                           resettingSC := #statUnitStatus.state.resetting AND NOT "Unit1.Em6.Alarms".emAlarms.error,
                           startingSC := #statUnitStatus.state.starting AND "Unit1.Em6.ControlNodes".em.status.initialized AND "Unit1.Em6.ControlNodes".em.status.homed AND "Unit1.EmNodes".stateCommandsExecute,
                           stoppingSC := #statUnitStatus.state.stopping AND NOT #instHotPressLeftHomeJob1.jobStatus.active AND NOT #instHotPressLeftLoadJob2.jobStatus.active AND NOT #instHotPressLeftInspectionJob3.jobStatus.active AND NOT #instHotPressLeftUnloadJob4.jobStatus.active,
                           abortingSC := #statUnitStatus.state.aborting AND #TRUE,
                           clearingSC := #statUnitStatus.state.clearing AND #TRUE,
                           holdingSC := #statUnitStatus.state.holding AND #TRUE,
                           unholdingSC := #statUnitStatus.state.unholding AND #TRUE,
                           suspendingSC := #statUnitStatus.state.suspending AND #TRUE,
                           unsuspendingSC := #statUnitStatus.state.unsuspending AND #TRUE,
                           completingSC := #statUnitStatus.state.completing AND NOT #instHotPressLeftHomeJob1.jobStatus.active AND NOT #instHotPressLeftLoadJob2.jobStatus.active AND NOT #instHotPressLeftInspectionJob3.jobStatus.active AND NOT #instHotPressLeftUnloadJob4.jobStatus.active,
                           stateComplete => #tempScInProduction);
END_REGION

REGION Network 62: Determine StateComplete (SC) in Mode Maintenance/Manual
   // Conditions for the Equipment Modules "stateComplete" feedback to the unit. This feedback is given when the task in for the respective state is complete.
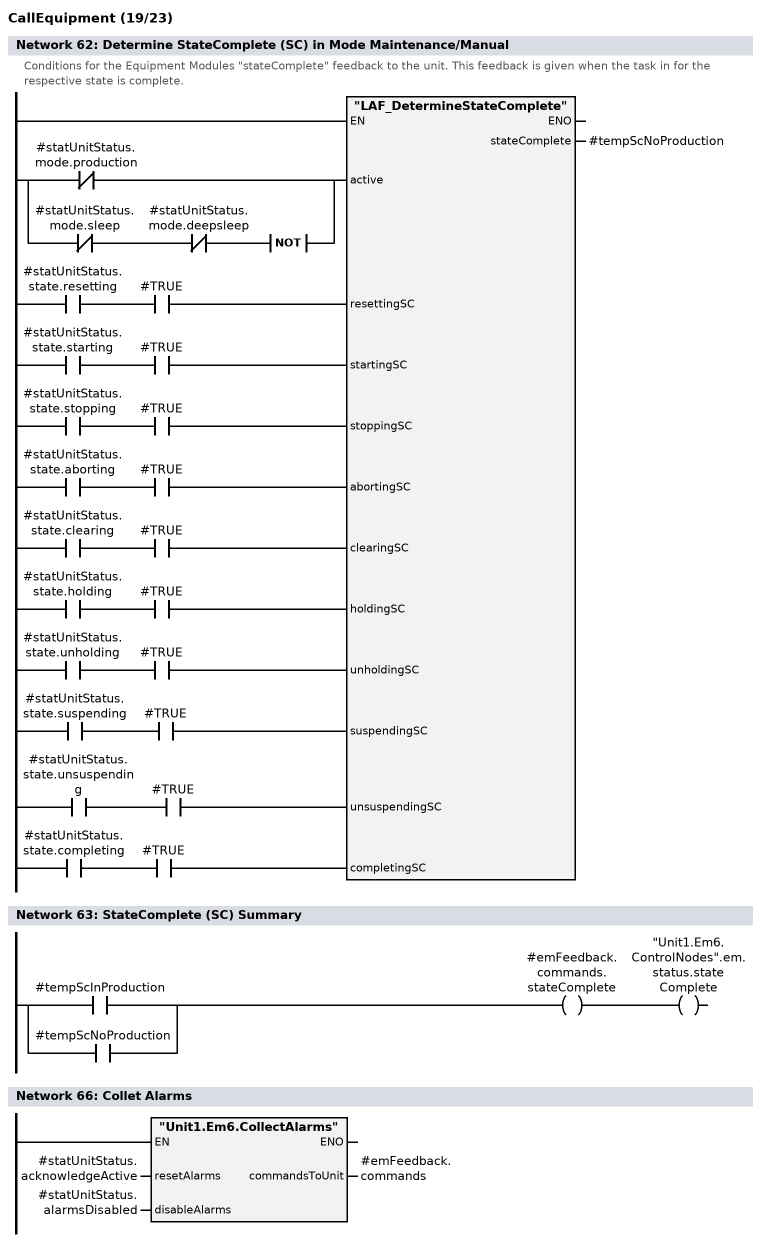
   RUNG wire#powerrail
      "LAF_DetermineStateComplete"(active := wire#w1, resettingSC := wire#w2, startingSC := wire#w3, stoppingSC := wire#w4, abortingSC := wire#w5, clearingSC := wire#w6, holdingSC := wire#w7, unholdingSC := wire#w8, suspendingSC := wire#w9, unsuspendingSC := wire#w10, completingSC := wire#w11, stateComplete => #tempScNoProduction)
   END_RUNG
   RUNG wire#powerrail
      I_Contact( #statUnitStatus.mode.production )
   END_RUNG wire#w1
   RUNG wire#powerrail
      I_Contact( #statUnitStatus.mode.sleep )
      I_Contact( #statUnitStatus.mode.deepsleep )
      Not()
   END_RUNG wire#w1
   RUNG wire#powerrail
      Contact( #statUnitStatus.state.resetting )
      Contact( #TRUE )
   END_RUNG wire#w2
   RUNG wire#powerrail
      Contact( #statUnitStatus.state.starting )
      Contact( #TRUE )
   END_RUNG wire#w3
   RUNG wire#powerrail
      Contact( #statUnitStatus.state.stopping )
      Contact( #TRUE )
   END_RUNG wire#w4
   RUNG wire#powerrail
      Contact( #statUnitStatus.state.aborting )
      Contact( #TRUE )
   END_RUNG wire#w5
   RUNG wire#powerrail
      Contact( #statUnitStatus.state.clearing )
      Contact( #TRUE )
   END_RUNG wire#w6
   RUNG wire#powerrail
      Contact( #statUnitStatus.state.holding )
      Contact( #TRUE )
   END_RUNG wire#w7
   RUNG wire#powerrail
      Contact( #statUnitStatus.state.unholding )
      Contact( #TRUE )
   END_RUNG wire#w8
   RUNG wire#powerrail
      Contact( #statUnitStatus.state.suspending )
      Contact( #TRUE )
   END_RUNG wire#w9
   RUNG wire#powerrail
      Contact( #statUnitStatus.state.unsuspending )
      Contact( #TRUE )
   END_RUNG wire#w10
   RUNG wire#powerrail
      Contact( #statUnitStatus.state.completing )
      Contact( #TRUE )
   END_RUNG wire#w11
   // the same network as SCL:
   "LAF_DetermineStateComplete"(active := NOT #statUnitStatus.mode.production OR NOT (NOT #statUnitStatus.mode.sleep AND NOT #statUnitStatus.mode.deepsleep),
                           resettingSC := #statUnitStatus.state.resetting AND #TRUE,
                           startingSC := #statUnitStatus.state.starting AND #TRUE,
                           stoppingSC := #statUnitStatus.state.stopping AND #TRUE,
                           abortingSC := #statUnitStatus.state.aborting AND #TRUE,
                           clearingSC := #statUnitStatus.state.clearing AND #TRUE,
                           holdingSC := #statUnitStatus.state.holding AND #TRUE,
                           unholdingSC := #statUnitStatus.state.unholding AND #TRUE,
                           suspendingSC := #statUnitStatus.state.suspending AND #TRUE,
                           unsuspendingSC := #statUnitStatus.state.unsuspending AND #TRUE,
                           completingSC := #statUnitStatus.state.completing AND #TRUE,
                           stateComplete => #tempScNoProduction);
END_REGION

REGION Network 63: StateComplete (SC) Summary
   RUNG wire#powerrail
      Contact( #tempScInProduction )
      wire#w1
      Coil( #emFeedback.commands.stateComplete )
      Coil( "Unit1.Em6.ControlNodes".em.status.stateComplete )
   END_RUNG
   RUNG wire#powerrail
      Contact( #tempScNoProduction )
   END_RUNG wire#w1
   // the same network as SCL:
   #emFeedback.commands.stateComplete := #tempScInProduction OR #tempScNoProduction;
   "Unit1.Em6.ControlNodes".em.status.stateComplete := #emFeedback.commands.stateComplete;
END_REGION

REGION Network 65: ******************** Alarms ********************
END_REGION

REGION Network 66: Collet Alarms
   RUNG wire#powerrail
      "Unit1.Em6.CollectAlarms"(resetAlarms := #statUnitStatus.acknowledgeActive, disableAlarms := #statUnitStatus.alarmsDisabled, commandsToUnit => #emFeedback.commands)
   END_RUNG
   // the same network as SCL:
   "Unit1.Em6.CollectAlarms"(resetAlarms := #statUnitStatus.acknowledgeActive,
                           disableAlarms := #statUnitStatus.alarmsDisabled,
                           commandsToUnit => #emFeedback.commands);
END_REGION

REGION Network 67: Manage Alarms
   // Derive commands from the ProDiag supervision. The ProDiag supervisions contain categories which define the reaction of these supervisions (e.g. abort, stop, hold). These are handed over as commands to the unit level.
   // Alternatively, if no ProDiag should be used, you can use the LAF_ManageBitAlarms to realize bit alarm handling. This block can be found in LAF in folder 70_AlarmHandling.
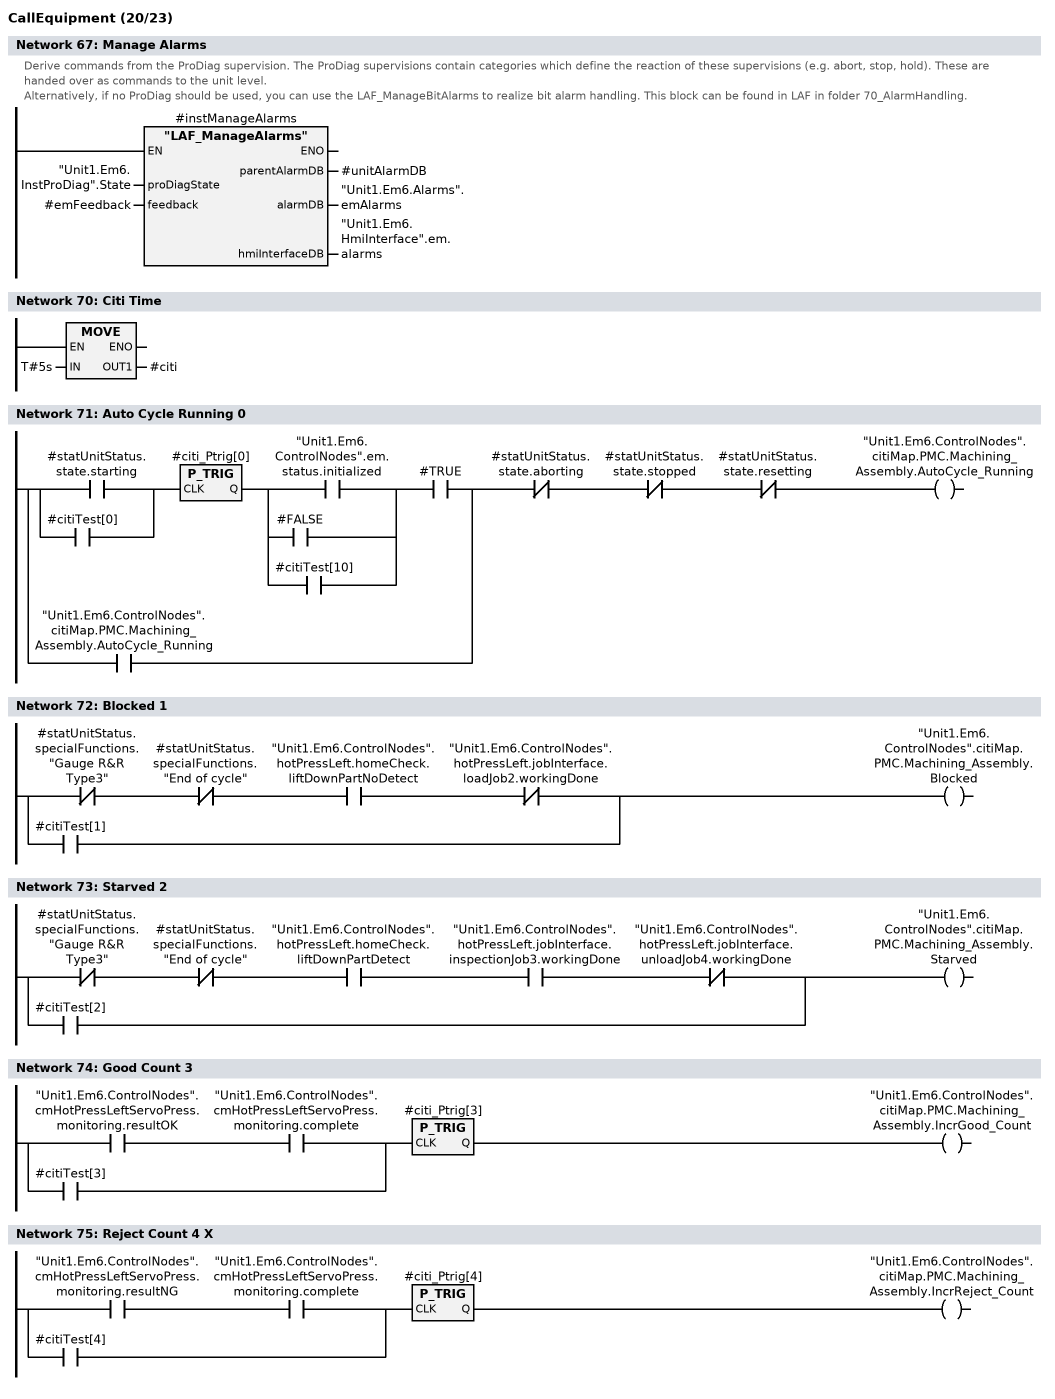
   RUNG wire#powerrail
      #instManageAlarms(proDiagState := "Unit1.Em6.InstProDiag".State, feedback := #emFeedback, parentAlarmDB => #unitAlarmDB, alarmDB => "Unit1.Em6.Alarms".emAlarms, hmiInterfaceDB => "Unit1.Em6.HmiInterface".em.alarms)
   END_RUNG
   // the same network as SCL:
   #instManageAlarms(proDiagState := "Unit1.Em6.InstProDiag".State,   // "LAF_ManageAlarms"
                     feedback := #emFeedback,
                     parentAlarmDB => #unitAlarmDB,
                     alarmDB => "Unit1.Em6.Alarms".emAlarms,
                     hmiInterfaceDB => "Unit1.Em6.HmiInterface".em.alarms);
END_REGION

REGION Network 69: ******************** CITI ********************
END_REGION

REGION Network 70: Citi Time
   RUNG wire#powerrail
      Move(in := T#5s, out1 => #citi)
   END_RUNG
   // the same network as SCL:
   #citi := T#5s;
END_REGION

REGION Network 71: Auto Cycle Running 0
   RUNG wire#powerrail
      Contact( #statUnitStatus.state.starting )
      wire#w1
      P_Trig( #citi_Ptrig[0] )
      wire#w2
      Contact( "Unit1.Em6.ControlNodes".em.status.initialized )
      wire#w3
      Contact( #TRUE )
      wire#w4
      I_Contact( #statUnitStatus.state.aborting )
      I_Contact( #statUnitStatus.state.stopped )
      I_Contact( #statUnitStatus.state.resetting )
      Coil( "Unit1.Em6.ControlNodes".citiMap.PMC.Machining_Assembly.AutoCycle_Running )
   END_RUNG
   RUNG wire#powerrail
      Contact( #citiTest[0] )
   END_RUNG wire#w1
   RUNG wire#w2
      Contact( #FALSE )
   END_RUNG wire#w3
   RUNG wire#w2
      Contact( #citiTest[10] )
   END_RUNG wire#w3
   RUNG wire#powerrail
      Contact( "Unit1.Em6.ControlNodes".citiMap.PMC.Machining_Assembly.AutoCycle_Running )
   END_RUNG wire#w4
   // the same network as SCL:
   #_w1 := #statUnitStatus.state.starting OR #citiTest[0];
   #_w2 := #_w1 AND NOT #citi_Ptrig[0];   // rising edge
   #citi_Ptrig[0] := #_w1;
   "Unit1.Em6.ControlNodes".citiMap.PMC.Machining_Assembly.AutoCycle_Running := ((#_w2 AND ("Unit1.Em6.ControlNodes".em.status.initialized OR #FALSE OR #citiTest[10]) AND #TRUE) OR "Unit1.Em6.ControlNodes".citiMap.PMC.Machining_Assembly.AutoCycle_Running) AND NOT #statUnitStatus.state.aborting AND NOT #statUnitStatus.state.stopped AND NOT #statUnitStatus.state.resetting;
END_REGION

REGION Network 72: Blocked 1
   RUNG wire#powerrail
      I_Contact( #statUnitStatus.specialFunctions."Gauge R&R Type3" )
      I_Contact( #statUnitStatus.specialFunctions."End of cycle" )
      Contact( "Unit1.Em6.ControlNodes".hotPressLeft.homeCheck.liftDownPartNoDetect )
      I_Contact( "Unit1.Em6.ControlNodes".hotPressLeft.jobInterface.loadJob2.workingDone )
      wire#w1
      Coil( "Unit1.Em6.ControlNodes".citiMap.PMC.Machining_Assembly.Blocked )
   END_RUNG
   RUNG wire#powerrail
      Contact( #citiTest[1] )
   END_RUNG wire#w1
   // the same network as SCL:
   "Unit1.Em6.ControlNodes".citiMap.PMC.Machining_Assembly.Blocked := (NOT #statUnitStatus.specialFunctions."Gauge R&R Type3" AND NOT #statUnitStatus.specialFunctions."End of cycle" AND "Unit1.Em6.ControlNodes".hotPressLeft.homeCheck.liftDownPartNoDetect AND NOT "Unit1.Em6.ControlNodes".hotPressLeft.jobInterface.loadJob2.workingDone) OR #citiTest[1];
END_REGION

REGION Network 73: Starved 2
   RUNG wire#powerrail
      I_Contact( #statUnitStatus.specialFunctions."Gauge R&R Type3" )
      I_Contact( #statUnitStatus.specialFunctions."End of cycle" )
      Contact( "Unit1.Em6.ControlNodes".hotPressLeft.homeCheck.liftDownPartDetect )
      Contact( "Unit1.Em6.ControlNodes".hotPressLeft.jobInterface.inspectionJob3.workingDone )
      I_Contact( "Unit1.Em6.ControlNodes".hotPressLeft.jobInterface.unloadJob4.workingDone )
      wire#w1
      Coil( "Unit1.Em6.ControlNodes".citiMap.PMC.Machining_Assembly.Starved )
   END_RUNG
   RUNG wire#powerrail
      Contact( #citiTest[2] )
   END_RUNG wire#w1
   // the same network as SCL:
   "Unit1.Em6.ControlNodes".citiMap.PMC.Machining_Assembly.Starved := (NOT #statUnitStatus.specialFunctions."Gauge R&R Type3" AND NOT #statUnitStatus.specialFunctions."End of cycle" AND "Unit1.Em6.ControlNodes".hotPressLeft.homeCheck.liftDownPartDetect AND "Unit1.Em6.ControlNodes".hotPressLeft.jobInterface.inspectionJob3.workingDone AND NOT "Unit1.Em6.ControlNodes".hotPressLeft.jobInterface.unloadJob4.workingDone) OR #citiTest[2];
END_REGION

